NETWORK
TITLE = T-10.00 DOSE ON OFF
      O     "Blend to Preparation"."T-20".Raw_Material.Vinegar.DoseRun;
      O     "Blend to Preparation"."T-21".Raw_Material.Vinegar.DoseRun;
      O     "Blend to Preparation"."T-30".Raw_Material.Vinegar.DoseRun;
      O     "Blend to Preparation"."T-31".Raw_Material.Vinegar.DoseRun;
      O     "Blend to Preparation"."T-40".Raw_Material.Vinegar.DoseRun;
      O     "Blend to Preparation"."T-41".Raw_Material.Vinegar.DoseRun;
      O     "T-05_Tomato"."Vinegar Req";

      =     "T-10_Vinegar".IN_Dose_Run;

NETWORK
TITLE = T-10.00 DOSE PAUSE
      O     "Blend to Preparation"."T-20".Raw_Material.Vinegar.DoseHeld;
      O     "Blend to Preparation"."T-21".Raw_Material.Vinegar.DoseHeld;
      O     "Blend to Preparation"."T-30".Raw_Material.Vinegar.DoseHeld;
      O     "Blend to Preparation"."T-31".Raw_Material.Vinegar.DoseHeld;
      O     "Blend to Preparation"."T-40".Raw_Material.Vinegar.DoseHeld;
      O     "Blend to Preparation"."T-41".Raw_Material.Vinegar.DoseHeld;
      O     "T-05_Tomato".Dose_Vinegar.QHELD;

      =     "T-10_Vinegar".IN_Dose_Held;

NETWORK
TITLE = T-10.00 DOSE VALVE CMD
      O(;
      A     "Blend to Preparation"."T-20".Raw_Material.Vinegar.DoseRun;
      A     "Blend to Preparation"."T-20".Raw_Material.Vinegar.ValveCMD;
      );
      O(;
      A     "Blend to Preparation"."T-21".Raw_Material.Vinegar.DoseRun;
      A     "Blend to Preparation"."T-21".Raw_Material.Vinegar.ValveCMD;
      );
      O(;
      A     "Blend to Preparation"."T-30".Raw_Material.Vinegar.DoseRun;
      A     "Blend to Preparation"."T-30".Raw_Material.Vinegar.ValveCMD;
      );
      O(;
      A     "Blend to Preparation"."T-31".Raw_Material.Vinegar.DoseRun;
      A     "Blend to Preparation"."T-31".Raw_Material.Vinegar.ValveCMD;
      );
      O(;
      A     "Blend to Preparation"."T-40".Raw_Material.Vinegar.DoseRun;
      A     "Blend to Preparation"."T-40".Raw_Material.Vinegar.ValveCMD;
      );
      O(;
      A     "Blend to Preparation"."T-41".Raw_Material.Vinegar.DoseRun;
      A     "Blend to Preparation"."T-41".Raw_Material.Vinegar.ValveCMD;
      );
      O(;
      A     "T-05_Tomato"."Vinegar Req";
      A     "T-05_Tomato".Dose_Vinegar.V_CMD;
      );

      =     "T-10_Vinegar".IN_Dose_Valve_Cmd;



NETWORK
TITLE = T-10.00 DOSE Pump CMD
      O(;
      A     "Blend to Preparation"."T-20".Raw_Material.Vinegar.DoseRun;
      A     "Blend to Preparation"."T-20".Raw_Material.Vinegar.PumpCMD;
      );
      O(;
      A     "Blend to Preparation"."T-21".Raw_Material.Vinegar.DoseRun;
      A     "Blend to Preparation"."T-21".Raw_Material.Vinegar.PumpCMD;
      );
      O(;
      A     "Blend to Preparation"."T-30".Raw_Material.Vinegar.DoseRun;
      A     "Blend to Preparation"."T-30".Raw_Material.Vinegar.PumpCMD;
      );
      O(;
      A     "Blend to Preparation"."T-31".Raw_Material.Vinegar.DoseRun;
      A     "Blend to Preparation"."T-31".Raw_Material.Vinegar.PumpCMD;
      );
      O(;
      A     "Blend to Preparation"."T-40".Raw_Material.Vinegar.DoseRun;
      A     "Blend to Preparation"."T-40".Raw_Material.Vinegar.PumpCMD;
      );
      O(;
      A     "Blend to Preparation"."T-41".Raw_Material.Vinegar.DoseRun;
      A     "Blend to Preparation"."T-41".Raw_Material.Vinegar.PumpCMD;
      );
      O(;
      A     "T-05_Tomato"."Vinegar Req";
      A     "T-05_Tomato".Dose_Vinegar.P_CMD;
      );

      =     "T-10_Vinegar".IN_Dose_Pump_Cmd;



NETWORK
TITLE = T-10.00 DOSE PUMP SPEED
// Checking
      O     "Blend to Preparation"."T-20".Raw_Material.Vinegar.DoseRun;
      JC    SP_10_FROM_20;
      O     "Blend to Preparation"."T-21".Raw_Material.Vinegar.DoseRun;
      JC    SP_10_FROM_21;
      O     "Blend to Preparation"."T-30".Raw_Material.Vinegar.DoseRun;
      JC    SP_10_FROM_30;
      O     "Blend to Preparation"."T-31".Raw_Material.Vinegar.DoseRun;
      JC    SP_10_FROM_31;
      O     "Blend to Preparation"."T-40".Raw_Material.Vinegar.DoseRun;
      JC    SP_10_FROM_40;
      O     "Blend to Preparation"."T-41".Raw_Material.Vinegar.DoseRun;
      JC    SP_10_FROM_41;
      O     "T-05_Tomato"."Vinegar Req";
      JC    SP_10_FROM_Tomato;

//Jump to end if Blend not Dosing
      JC    SP_10_SELF;
//Load Set Point
SP_10_FROM_20:L     "Blend to Preparation".Recipe."T-20".Vinegar.SP_PumpSpeed;
      T     "T-10_Vinegar".IN_Dose_Pump_Sp;
      JC    SP_10_SELF;
SP_10_FROM_21:L     "Blend to Preparation".Recipe."T-21".Vinegar.SP_PumpSpeed;
      T     "T-10_Vinegar".IN_Dose_Pump_Sp;
      JC    SP_10_SELF;
SP_10_FROM_30:L     "Blend to Preparation".Recipe."T-30".Vinegar.SP_PumpSpeed;
      T     "T-10_Vinegar".IN_Dose_Pump_Sp;
      JC    SP_10_SELF;
SP_10_FROM_31:L     "Blend to Preparation".Recipe."T-31".Vinegar.SP_PumpSpeed;
      T     "T-10_Vinegar".IN_Dose_Pump_Sp;
      JC    SP_10_SELF;
SP_10_FROM_40:L     "Blend to Preparation".Recipe."T-40".Vinegar.SP_PumpSpeed;
      T     "T-10_Vinegar".IN_Dose_Pump_Sp;
      JC    SP_10_SELF;
SP_10_FROM_41:L     "Blend to Preparation".Recipe."T-41".Vinegar.SP_PumpSpeed;
      T     "T-10_Vinegar".IN_Dose_Pump_Sp;
      JC    SP_10_SELF;
SP_10_FROM_Tomato:L     "T-05_Tomato".Dose_Vinegar.P_SPEED;
      T     "T-10_Vinegar".IN_Dose_Pump_Sp;
      JC    SP_10_SELF;

// END
SP_10_SELF:L     "T-10_Vinegar".IN_Dose_Pump_Sp;
      T     "T-10_Vinegar".IN_Dose_Pump_Sp;


REGION Network 130: T-010.00 LineTransferOK
   RUNG wire#powerrail
      Contact( "AlwaysTRUE" )
      wire#w1
      Contact( "Blend to Preparation"."T-20".LineVinegar_OK )
      wire#w2
      Coil( "T-10_Vinegar".IN_Dose_LineOK )
   END_RUNG
   RUNG wire#w1
      Contact( "Blend to Preparation"."T-21".LineVinegar_OK )
   END_RUNG wire#w2
   RUNG wire#w1
      Contact( "Blend to Preparation"."T-30".LineVinegar_OK )
   END_RUNG wire#w2
   RUNG wire#w1
      Contact( "Blend to Preparation"."T-31".LineVinegar_OK )
   END_RUNG wire#w2
   RUNG wire#w1
      Contact( "Blend to Preparation"."T-40".LineVinegar_OK )
   END_RUNG wire#w2
   RUNG wire#w1
      Contact( "Blend to Preparation"."T-41".LineVinegar_OK )
   END_RUNG wire#w2
   RUNG wire#w1
      Contact( "T-05_Tomato".IN_FBAV_Vinegar )
   END_RUNG wire#w2
   // the same network as SCL:
   "T-10_Vinegar".IN_Dose_LineOK := "AlwaysTRUE" AND ("Blend to Preparation"."T-20".LineVinegar_OK OR "Blend to Preparation"."T-21".LineVinegar_OK OR "Blend to Preparation"."T-30".LineVinegar_OK OR "Blend to Preparation"."T-31".LineVinegar_OK OR "Blend to Preparation"."T-40".LineVinegar_OK OR "Blend to Preparation"."T-41".LineVinegar_OK OR "T-05_Tomato".IN_FBAV_Vinegar);
END_REGION

REGION Network 131: T-10.00____VINEGAR
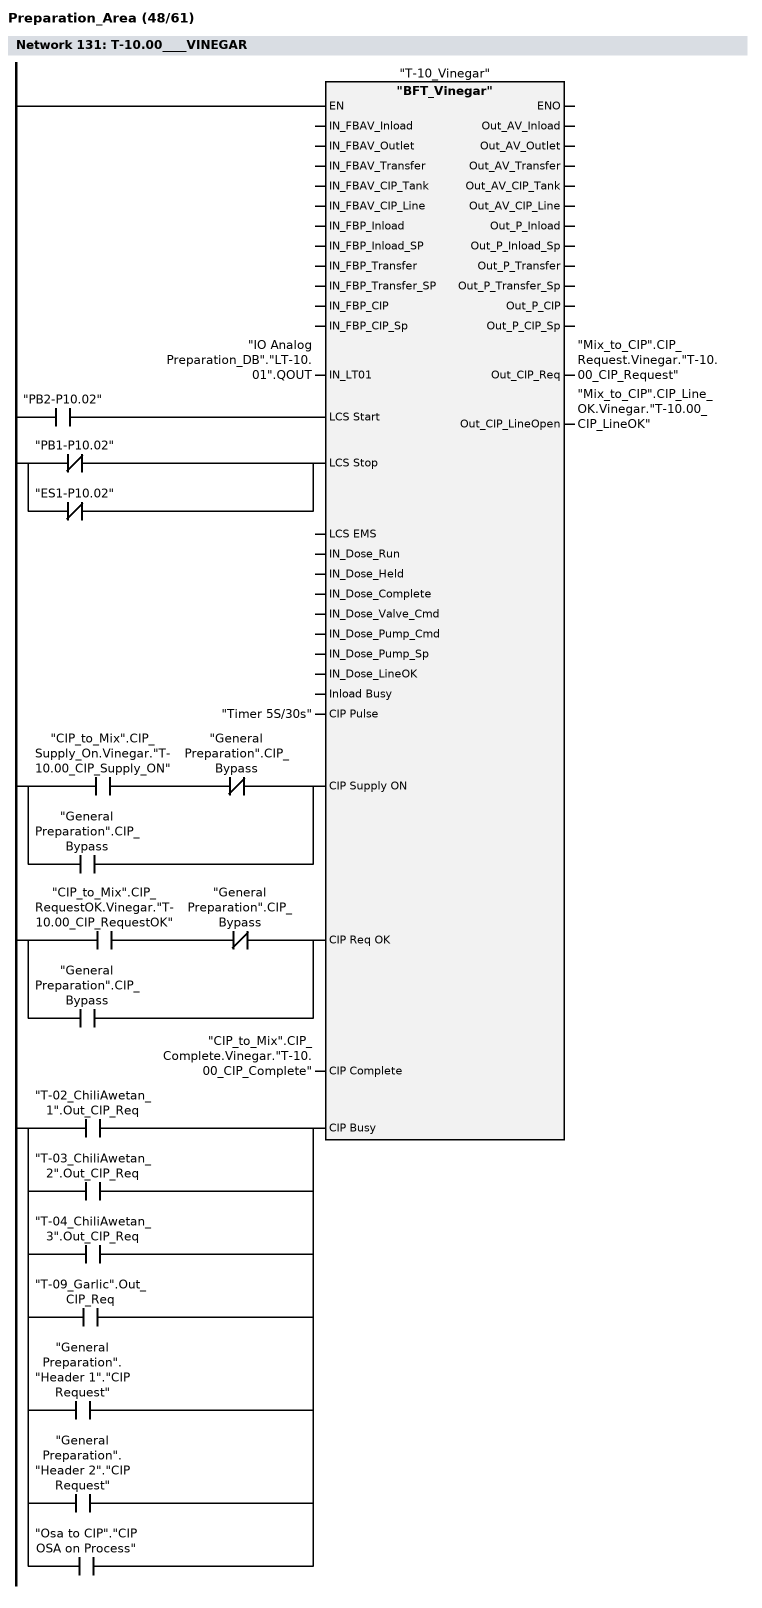
   RUNG wire#powerrail
      "T-10_Vinegar"("LCS Start" := wire#w1, "LCS Stop" := wire#w2, "CIP Supply ON" := wire#w3, "CIP Req OK" := wire#w4, "CIP Busy" := wire#w5, IN_FBAV_Inload :=, IN_FBAV_Outlet :=, IN_FBAV_Transfer :=, IN_FBAV_CIP_Tank :=, IN_FBAV_CIP_Line :=, IN_FBP_Inload :=, IN_FBP_Inload_SP :=, IN_FBP_Transfer :=, IN_FBP_Transfer_SP :=, IN_FBP_CIP :=, IN_FBP_CIP_Sp :=, IN_LT01 := "IO Analog Preparation_DB"."LT-10.01".QOUT, "LCS EMS" :=, IN_Dose_Run :=, IN_Dose_Held :=, IN_Dose_Complete :=, IN_Dose_Valve_Cmd :=, IN_Dose_Pump_Cmd :=, IN_Dose_Pump_Sp :=, IN_Dose_LineOK :=, "Inload Busy" :=, "CIP Pulse" := "Timer 5S/30s", "CIP Complete" := "CIP_to_Mix".CIP_Complete.Vinegar."T-10.00_CIP_Complete", Out_AV_Inload =>, Out_AV_Outlet =>, Out_AV_Transfer =>, Out_AV_CIP_Tank =>, Out_AV_CIP_Line =>, Out_P_Inload =>, Out_P_Inload_Sp =>, Out_P_Transfer =>, Out_P_Transfer_Sp =>, Out_P_CIP =>, Out_P_CIP_Sp =>, Out_CIP_Req => "Mix_to_CIP".CIP_Request.Vinegar."T-10.00_CIP_Request", Out_CIP_LineOpen => "Mix_to_CIP".CIP_Line_OK.Vinegar."T-10.00_CIP_LineOK")
   END_RUNG
   RUNG wire#powerrail
      Contact( "PB2-P10.02" )
   END_RUNG wire#w1
   RUNG wire#powerrail
      I_Contact( "PB1-P10.02" )
   END_RUNG wire#w2
   RUNG wire#powerrail
      I_Contact( "ES1-P10.02" )
   END_RUNG wire#w2
   RUNG wire#powerrail
      Contact( "CIP_to_Mix".CIP_Supply_On.Vinegar."T-10.00_CIP_Supply_ON" )
      I_Contact( "General Preparation".CIP_Bypass )
   END_RUNG wire#w3
   RUNG wire#powerrail
      Contact( "General Preparation".CIP_Bypass )
   END_RUNG wire#w3
   RUNG wire#powerrail
      Contact( "CIP_to_Mix".CIP_RequestOK.Vinegar."T-10.00_CIP_RequestOK" )
      I_Contact( "General Preparation".CIP_Bypass )
   END_RUNG wire#w4
   RUNG wire#powerrail
      Contact( "General Preparation".CIP_Bypass )
   END_RUNG wire#w4
   RUNG wire#powerrail
      Contact( "T-02_ChiliAwetan_1".Out_CIP_Req )
   END_RUNG wire#w5
   RUNG wire#powerrail
      Contact( "T-03_ChiliAwetan_2".Out_CIP_Req )
   END_RUNG wire#w5
   RUNG wire#powerrail
      Contact( "T-04_ChiliAwetan_3".Out_CIP_Req )
   END_RUNG wire#w5
   RUNG wire#powerrail
      Contact( "T-09_Garlic".Out_CIP_Req )
   END_RUNG wire#w5
   RUNG wire#powerrail
      Contact( "General Preparation"."Header 1"."CIP Request" )
   END_RUNG wire#w5
   RUNG wire#powerrail
      Contact( "General Preparation"."Header 2"."CIP Request" )
   END_RUNG wire#w5
   RUNG wire#powerrail
      Contact( "Osa to CIP"."CIP OSA on Process" )
   END_RUNG wire#w5
   // the same network as SCL:
   "T-10_Vinegar"(IN_LT01 := "IO Analog Preparation_DB"."LT-10.01".QOUT,   // "BFT_Vinegar"
                  "LCS Start" := "PB2-P10.02",
                  "LCS Stop" := NOT "PB1-P10.02" OR NOT "ES1-P10.02",
                  "CIP Pulse" := "Timer 5S/30s",
                  "CIP Supply ON" := ("CIP_to_Mix".CIP_Supply_On.Vinegar."T-10.00_CIP_Supply_ON" AND NOT "General Preparation".CIP_Bypass) OR "General Preparation".CIP_Bypass,
                  "CIP Req OK" := ("CIP_to_Mix".CIP_RequestOK.Vinegar."T-10.00_CIP_RequestOK" AND NOT "General Preparation".CIP_Bypass) OR "General Preparation".CIP_Bypass,
                  "CIP Complete" := "CIP_to_Mix".CIP_Complete.Vinegar."T-10.00_CIP_Complete",
                  "CIP Busy" := "T-02_ChiliAwetan_1".Out_CIP_Req OR "T-03_ChiliAwetan_2".Out_CIP_Req OR "T-04_ChiliAwetan_3".Out_CIP_Req OR "T-09_Garlic".Out_CIP_Req OR "General Preparation"."Header 1"."CIP Request" OR "General Preparation"."Header 2"."CIP Request" OR "Osa to CIP"."CIP OSA on Process",
                  Out_CIP_Req => "Mix_to_CIP".CIP_Request.Vinegar."T-10.00_CIP_Request",
                  Out_CIP_LineOpen => "Mix_to_CIP".CIP_Line_OK.Vinegar."T-10.00_CIP_LineOK");
END_REGION

REGION Network 132: T-10.00 Valve Cmd
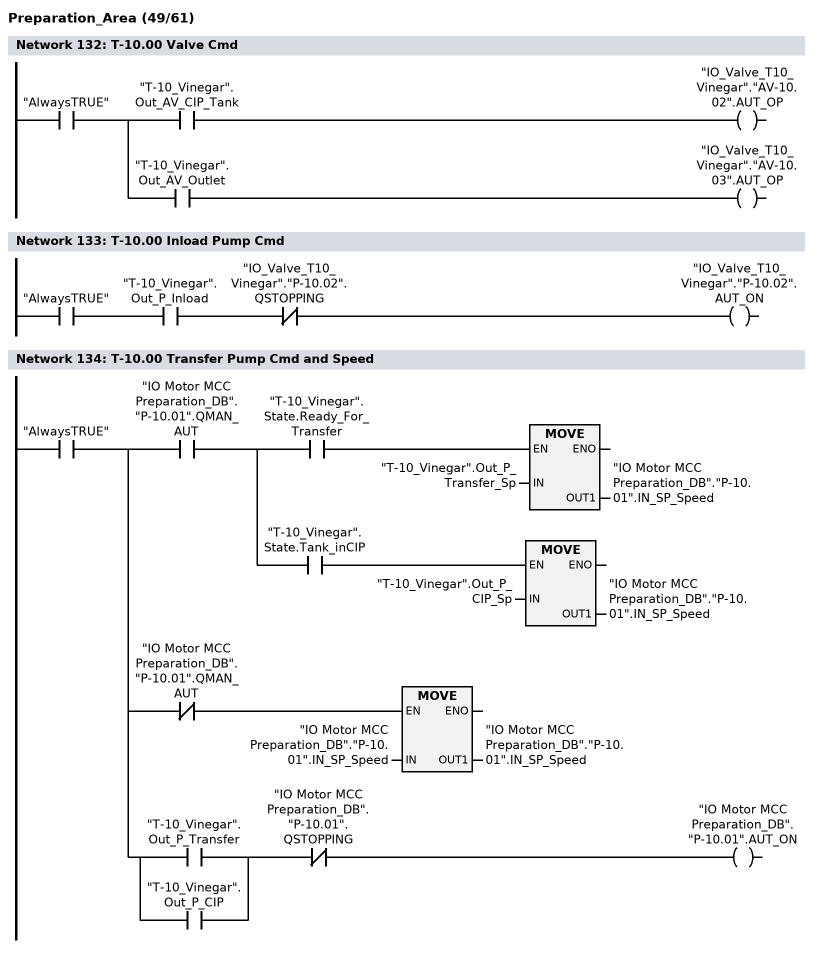
   RUNG wire#powerrail
      Contact( "AlwaysTRUE" )
      wire#w1
      Contact( "T-10_Vinegar".Out_AV_CIP_Tank )
      Coil( "IO_Valve_T10_Vinegar"."AV-10.02".AUT_OP )
   END_RUNG
   RUNG wire#w1
      Contact( "T-10_Vinegar".Out_AV_Outlet )
      Coil( "IO_Valve_T10_Vinegar"."AV-10.03".AUT_OP )
   END_RUNG
   // the same network as SCL:
   "IO_Valve_T10_Vinegar"."AV-10.02".AUT_OP := "AlwaysTRUE" AND "T-10_Vinegar".Out_AV_CIP_Tank;
   "IO_Valve_T10_Vinegar"."AV-10.03".AUT_OP := "AlwaysTRUE" AND "T-10_Vinegar".Out_AV_Outlet;
END_REGION

REGION Network 133: T-10.00 Inload Pump Cmd
   RUNG wire#powerrail
      Contact( "AlwaysTRUE" )
      Contact( "T-10_Vinegar".Out_P_Inload )
      I_Contact( "IO_Valve_T10_Vinegar"."P-10.02".QSTOPPING )
      Coil( "IO_Valve_T10_Vinegar"."P-10.02".AUT_ON )
   END_RUNG
   // the same network as SCL:
   "IO_Valve_T10_Vinegar"."P-10.02".AUT_ON := "AlwaysTRUE" AND "T-10_Vinegar".Out_P_Inload AND NOT "IO_Valve_T10_Vinegar"."P-10.02".QSTOPPING;
END_REGION

REGION Network 134: T-10.00 Transfer Pump Cmd and Speed
   RUNG wire#powerrail
      Contact( "AlwaysTRUE" )
      wire#w1
      Contact( "IO Motor MCC Preparation_DB"."P-10.01".QMAN_AUT )
      wire#w2
      Contact( "T-10_Vinegar".State.Ready_For_Transfer )
      Move(in := "T-10_Vinegar".Out_P_Transfer_Sp, out1 => "IO Motor MCC Preparation_DB"."P-10.01".IN_SP_Speed)
   END_RUNG
   RUNG wire#w2
      Contact( "T-10_Vinegar".State.Tank_inCIP )
      Move(in := "T-10_Vinegar".Out_P_CIP_Sp, out1 => "IO Motor MCC Preparation_DB"."P-10.01".IN_SP_Speed)
   END_RUNG
   RUNG wire#w1
      I_Contact( "IO Motor MCC Preparation_DB"."P-10.01".QMAN_AUT )
      Move(in := "IO Motor MCC Preparation_DB"."P-10.01".IN_SP_Speed, out1 => "IO Motor MCC Preparation_DB"."P-10.01".IN_SP_Speed)
   END_RUNG
   RUNG wire#w1
      Contact( "T-10_Vinegar".Out_P_Transfer )
      wire#w3
      I_Contact( "IO Motor MCC Preparation_DB"."P-10.01".QSTOPPING )
      Coil( "IO Motor MCC Preparation_DB"."P-10.01".AUT_ON )
   END_RUNG
   RUNG wire#w1
      Contact( "T-10_Vinegar".Out_P_CIP )
   END_RUNG wire#w3
   // the same network as SCL:
   #_w1 := "AlwaysTRUE" AND "IO Motor MCC Preparation_DB"."P-10.01".QMAN_AUT;
   IF #_w1 AND "T-10_Vinegar".State.Ready_For_Transfer THEN
       "IO Motor MCC Preparation_DB"."P-10.01".IN_SP_Speed := "T-10_Vinegar".Out_P_Transfer_Sp;
   END_IF;
   IF #_w1 AND "T-10_Vinegar".State.Tank_inCIP THEN
       "IO Motor MCC Preparation_DB"."P-10.01".IN_SP_Speed := "T-10_Vinegar".Out_P_CIP_Sp;
   END_IF;
   IF "AlwaysTRUE" AND NOT "IO Motor MCC Preparation_DB"."P-10.01".QMAN_AUT THEN
       "IO Motor MCC Preparation_DB"."P-10.01".IN_SP_Speed := "IO Motor MCC Preparation_DB"."P-10.01".IN_SP_Speed;
   END_IF;
   "IO Motor MCC Preparation_DB"."P-10.01".AUT_ON := "AlwaysTRUE" AND ("T-10_Vinegar".Out_P_Transfer OR "T-10_Vinegar".Out_P_CIP) AND NOT "IO Motor MCC Preparation_DB"."P-10.01".QSTOPPING;
END_REGION

REGION Network 135: T-10.00 Feedback Instrument
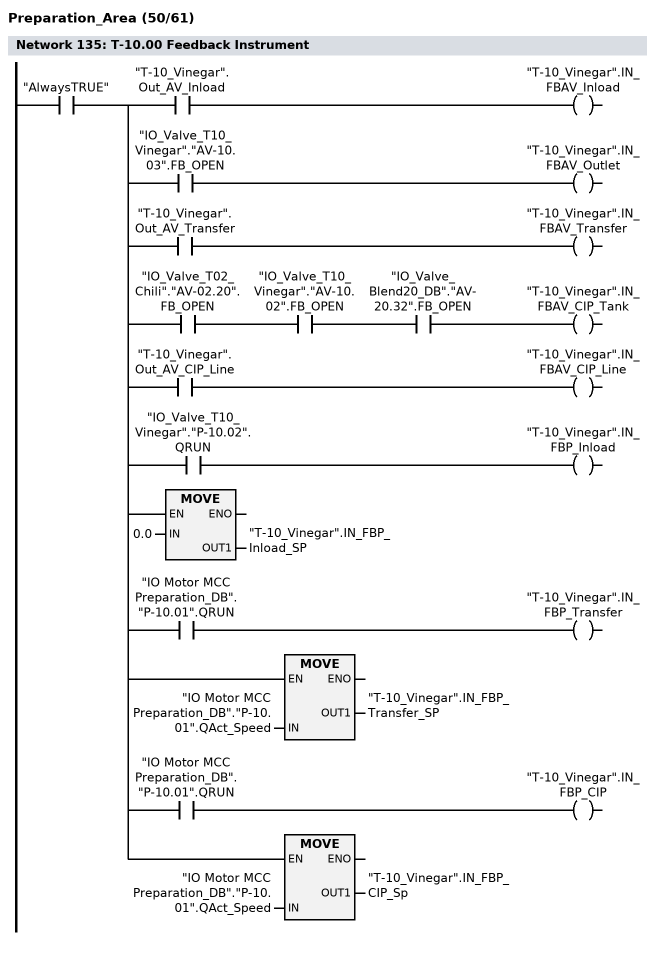
   RUNG wire#powerrail
      Contact( "AlwaysTRUE" )
      wire#w1
      Contact( "T-10_Vinegar".Out_AV_Inload )
      Coil( "T-10_Vinegar".IN_FBAV_Inload )
   END_RUNG
   RUNG wire#w1
      Contact( "IO_Valve_T10_Vinegar"."AV-10.03".FB_OPEN )
      Coil( "T-10_Vinegar".IN_FBAV_Outlet )
   END_RUNG
   RUNG wire#w1
      Contact( "T-10_Vinegar".Out_AV_Transfer )
      Coil( "T-10_Vinegar".IN_FBAV_Transfer )
   END_RUNG
   RUNG wire#w1
      Contact( "IO_Valve_T02_Chili"."AV-02.20".FB_OPEN )
      Contact( "IO_Valve_T10_Vinegar"."AV-10.02".FB_OPEN )
      Contact( "IO_Valve_Blend20_DB"."AV-20.32".FB_OPEN )
      Coil( "T-10_Vinegar".IN_FBAV_CIP_Tank )
   END_RUNG
   RUNG wire#w1
      Contact( "T-10_Vinegar".Out_AV_CIP_Line )
      Coil( "T-10_Vinegar".IN_FBAV_CIP_Line )
   END_RUNG
   RUNG wire#w1
      Contact( "IO_Valve_T10_Vinegar"."P-10.02".QRUN )
      Coil( "T-10_Vinegar".IN_FBP_Inload )
   END_RUNG
   RUNG wire#w1
      Move(in := 0.0, out1 => "T-10_Vinegar".IN_FBP_Inload_SP)
   END_RUNG
   RUNG wire#w1
      Contact( "IO Motor MCC Preparation_DB"."P-10.01".QRUN )
      Coil( "T-10_Vinegar".IN_FBP_Transfer )
   END_RUNG
   RUNG wire#w1
      Move(in := "IO Motor MCC Preparation_DB"."P-10.01".QAct_Speed, out1 => "T-10_Vinegar".IN_FBP_Transfer_SP)
   END_RUNG
   RUNG wire#w1
      Contact( "IO Motor MCC Preparation_DB"."P-10.01".QRUN )
      Coil( "T-10_Vinegar".IN_FBP_CIP )
   END_RUNG
   RUNG wire#w1
      Move(in := "IO Motor MCC Preparation_DB"."P-10.01".QAct_Speed, out1 => "T-10_Vinegar".IN_FBP_CIP_Sp)
   END_RUNG
   // the same network as SCL:
   "T-10_Vinegar".IN_FBAV_Inload := "AlwaysTRUE" AND "T-10_Vinegar".Out_AV_Inload;
   "T-10_Vinegar".IN_FBAV_Outlet := "AlwaysTRUE" AND "IO_Valve_T10_Vinegar"."AV-10.03".FB_OPEN;
   "T-10_Vinegar".IN_FBAV_Transfer := "AlwaysTRUE" AND "T-10_Vinegar".Out_AV_Transfer;
   "T-10_Vinegar".IN_FBAV_CIP_Tank := "AlwaysTRUE" AND "IO_Valve_T02_Chili"."AV-02.20".FB_OPEN AND "IO_Valve_T10_Vinegar"."AV-10.02".FB_OPEN AND "IO_Valve_Blend20_DB"."AV-20.32".FB_OPEN;
   "T-10_Vinegar".IN_FBAV_CIP_Line := "AlwaysTRUE" AND "T-10_Vinegar".Out_AV_CIP_Line;
   "T-10_Vinegar".IN_FBP_Inload := "AlwaysTRUE" AND "IO_Valve_T10_Vinegar"."P-10.02".QRUN;
   IF "AlwaysTRUE" THEN "T-10_Vinegar".IN_FBP_Inload_SP := 0.0; END_IF;
   "T-10_Vinegar".IN_FBP_Transfer := "AlwaysTRUE" AND "IO Motor MCC Preparation_DB"."P-10.01".QRUN;
   IF "AlwaysTRUE" THEN
       "T-10_Vinegar".IN_FBP_Transfer_SP := "IO Motor MCC Preparation_DB"."P-10.01".QAct_Speed;
   END_IF;
   "T-10_Vinegar".IN_FBP_CIP := "AlwaysTRUE" AND "IO Motor MCC Preparation_DB"."P-10.01".QRUN;
   IF "AlwaysTRUE" THEN
       "T-10_Vinegar".IN_FBP_CIP_Sp := "IO Motor MCC Preparation_DB"."P-10.01".QAct_Speed;
   END_IF;
END_REGION

REGION Network 136: T-10.00 Comm to Blend
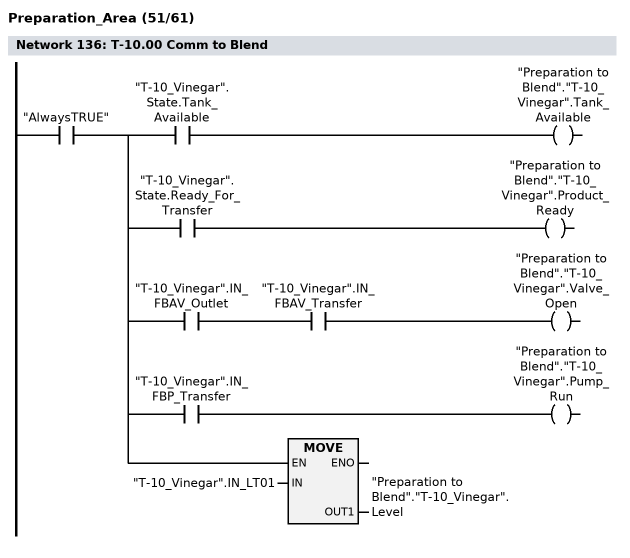
   RUNG wire#powerrail
      Contact( "AlwaysTRUE" )
      wire#w1
      Contact( "T-10_Vinegar".State.Tank_Available )
      Coil( "Preparation to Blend"."T-10_Vinegar".Tank_Available )
   END_RUNG
   RUNG wire#w1
      Contact( "T-10_Vinegar".State.Ready_For_Transfer )
      Coil( "Preparation to Blend"."T-10_Vinegar".Product_Ready )
   END_RUNG
   RUNG wire#w1
      Contact( "T-10_Vinegar".IN_FBAV_Outlet )
      Contact( "T-10_Vinegar".IN_FBAV_Transfer )
      Coil( "Preparation to Blend"."T-10_Vinegar".Valve_Open )
   END_RUNG
   RUNG wire#w1
      Contact( "T-10_Vinegar".IN_FBP_Transfer )
      Coil( "Preparation to Blend"."T-10_Vinegar".Pump_Run )
   END_RUNG
   RUNG wire#w1
      Move(in := "T-10_Vinegar".IN_LT01, out1 => "Preparation to Blend"."T-10_Vinegar".Level)
   END_RUNG
   // the same network as SCL:
   "Preparation to Blend"."T-10_Vinegar".Tank_Available := "AlwaysTRUE" AND "T-10_Vinegar".State.Tank_Available;
   "Preparation to Blend"."T-10_Vinegar".Product_Ready := "AlwaysTRUE" AND "T-10_Vinegar".State.Ready_For_Transfer;
   "Preparation to Blend"."T-10_Vinegar".Valve_Open := "AlwaysTRUE" AND "T-10_Vinegar".IN_FBAV_Outlet AND "T-10_Vinegar".IN_FBAV_Transfer;
   "Preparation to Blend"."T-10_Vinegar".Pump_Run := "AlwaysTRUE" AND "T-10_Vinegar".IN_FBP_Transfer;
   IF "AlwaysTRUE" THEN "Preparation to Blend"."T-10_Vinegar".Level := "T-10_Vinegar".IN_LT01; END_IF;
END_REGION

NETWORK
TITLE = T-51.00 DOSE ON OFF
      O     "Blend to Preparation"."T-20".Raw_Material.HW.DoseRun;
      O     "Blend to Preparation"."T-21".Raw_Material.HW.DoseRun;
      O     "Blend to Preparation"."T-30".Raw_Material.HW.DoseRun;
      O     "Blend to Preparation"."T-31".Raw_Material.HW.DoseRun;
      O     "Blend to Preparation"."T-40".Raw_Material.HW.DoseRun;
      O     "Blend to Preparation"."T-41".Raw_Material.HW.DoseRun;
      =     "T-51_HW".IN_Dose_Run;

NETWORK
TITLE = T-51.00 DOSE PAUSE
      O     "Blend to Preparation"."T-20".Raw_Material.HW.DoseHeld;
      O     "Blend to Preparation"."T-21".Raw_Material.HW.DoseHeld;
      O     "Blend to Preparation"."T-30".Raw_Material.HW.DoseHeld;
      O     "Blend to Preparation"."T-31".Raw_Material.HW.DoseHeld;
      O     "Blend to Preparation"."T-40".Raw_Material.HW.DoseHeld;
      O     "Blend to Preparation"."T-41".Raw_Material.HW.DoseHeld;
      =     "T-51_HW".IN_Dose_Held;

NETWORK
TITLE = T-51.00 DOSE VALVE CMD
      O(;
      A     "Blend to Preparation"."T-20".Raw_Material.HW.DoseRun;
      A     "Blend to Preparation"."T-20".Raw_Material.HW.ValveCMD;
      );
      O(;
      A     "Blend to Preparation"."T-21".Raw_Material.HW.DoseRun;
      A     "Blend to Preparation"."T-21".Raw_Material.HW.ValveCMD;
      );
      O(;
      A     "Blend to Preparation"."T-30".Raw_Material.HW.DoseRun;
      A     "Blend to Preparation"."T-30".Raw_Material.HW.ValveCMD;
      );
      O(;
      A     "Blend to Preparation"."T-31".Raw_Material.HW.DoseRun;
      A     "Blend to Preparation"."T-31".Raw_Material.HW.ValveCMD;
      );
      O(;
      A     "Blend to Preparation"."T-40".Raw_Material.HW.DoseRun;
      A     "Blend to Preparation"."T-40".Raw_Material.HW.ValveCMD;
      );
      O(;
      A     "Blend to Preparation"."T-41".Raw_Material.HW.DoseRun;
      A     "Blend to Preparation"."T-41".Raw_Material.HW.ValveCMD;
      );
      =     "T-51_HW".IN_Dose_Valve_Cmd;

NETWORK
TITLE = T-51.00 DOSE Pump CMD
      O(;
      A     "Blend to Preparation"."T-20".Raw_Material.HW.DoseRun;
      A     "Blend to Preparation"."T-20".Raw_Material.HW.PumpCMD;
      );
      O(;
      A     "Blend to Preparation"."T-21".Raw_Material.HW.DoseRun;
      A     "Blend to Preparation"."T-21".Raw_Material.HW.PumpCMD;
      );
      O(;
      A     "Blend to Preparation"."T-30".Raw_Material.HW.DoseRun;
      A     "Blend to Preparation"."T-30".Raw_Material.HW.PumpCMD;
      );
      O(;
      A     "Blend to Preparation"."T-31".Raw_Material.HW.DoseRun;
      A     "Blend to Preparation"."T-31".Raw_Material.HW.PumpCMD;
      );
      O(;
      A     "Blend to Preparation"."T-40".Raw_Material.HW.DoseRun;
      A     "Blend to Preparation"."T-40".Raw_Material.HW.PumpCMD;
      );
      O(;
      A     "Blend to Preparation"."T-41".Raw_Material.HW.DoseRun;
      A     "Blend to Preparation"."T-41".Raw_Material.HW.PumpCMD;
      );
      =     "T-51_HW".IN_Dose_Pump_Cmd;

NETWORK
TITLE = T-51.00 DOSE PUMP SPEED
// Checking
      O     "Blend to Preparation"."T-20".Raw_Material.HW.DoseRun;
      JC    SP_51_FROM_20;
      O     "Blend to Preparation"."T-21".Raw_Material.HW.DoseRun;
      JC    SP_51_FROM_21;
      O     "Blend to Preparation"."T-30".Raw_Material.HW.DoseRun;
      JC    SP_51_FROM_30;
      O     "Blend to Preparation"."T-31".Raw_Material.HW.DoseRun;
      JC    SP_51_FROM_31;
      O     "Blend to Preparation"."T-40".Raw_Material.HW.DoseRun;
      JC    SP_51_FROM_40;
      O     "Blend to Preparation"."T-41".Raw_Material.HW.DoseRun;
      JC    SP_51_FROM_41;
//Jump to end if Blend not Dosing
      JC    SP_51_SELF;
//Load Set Point
SP_51_FROM_20:L     "Blend to Preparation".Recipe."T-20".HW.SP_PumpSpeed;
      T     "T-51_HW".IN_Dose_Pump_Sp;
      JC    SP_51_SELF;
SP_51_FROM_21:L     "Blend to Preparation".Recipe."T-21".HW.SP_PumpSpeed;
      T     "T-51_HW".IN_Dose_Pump_Sp;
      JC    SP_51_SELF;
SP_51_FROM_30:L     "Blend to Preparation".Recipe."T-30".HW.SP_PumpSpeed;
      T     "T-51_HW".IN_Dose_Pump_Sp;
      JC    SP_51_SELF;
SP_51_FROM_31:L     "Blend to Preparation".Recipe."T-31".HW.SP_PumpSpeed;
      T     "T-51_HW".IN_Dose_Pump_Sp;
      JC    SP_51_SELF;
SP_51_FROM_40:L     "Blend to Preparation".Recipe."T-40".HW.SP_PumpSpeed;
      T     "T-51_HW".IN_Dose_Pump_Sp;
      JC    SP_51_SELF;
SP_51_FROM_41:L     "Blend to Preparation".Recipe."T-41".HW.SP_PumpSpeed;
      T     "T-51_HW".IN_Dose_Pump_Sp;
      JC    SP_51_SELF;
// END
SP_51_SELF:L     "T-51_HW".IN_Dose_Pump_Sp;
      T     "T-51_HW".IN_Dose_Pump_Sp;

NETWORK
TITLE = T-51.00 Header Req
// HEADER 1 Req
      O     "Blend to Preparation"."T-20".Raw_Material.HW.Header1_Req;
      O     "Blend to Preparation"."T-21".Raw_Material.HW.Header1_Req;
      O     "Blend to Preparation"."T-30".Raw_Material.HW.Header1_Req;
      O     "Blend to Preparation"."T-31".Raw_Material.HW.Header1_Req;
      O     "Blend to Preparation"."T-40".Raw_Material.HW.Header1_Req;
      O     "Blend to Preparation"."T-41".Raw_Material.HW.Header1_Req;
      =     "T-51_HW".IN_Dose_Header_1;

// HEADER 2 Req
      O     "Blend to Preparation"."T-20".Raw_Material.HW.Header2_Req;
      O     "Blend to Preparation"."T-21".Raw_Material.HW.Header2_Req;
      O     "Blend to Preparation"."T-30".Raw_Material.HW.Header2_Req;
      O     "Blend to Preparation"."T-31".Raw_Material.HW.Header2_Req;
      O     "Blend to Preparation"."T-40".Raw_Material.HW.Header2_Req;
      O     "Blend to Preparation"."T-41".Raw_Material.HW.Header2_Req;
      =     "T-51_HW".IN_Dose_Header_2;

REGION Network 145: T-51.00 LineTransferOK
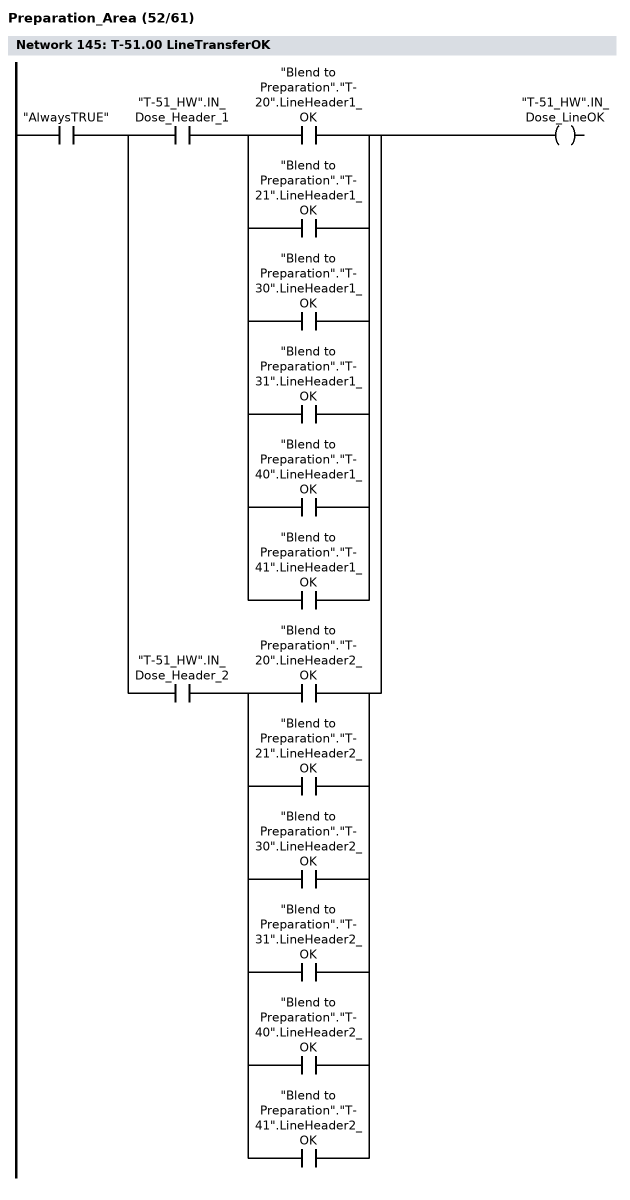
   RUNG wire#powerrail
      Contact( "AlwaysTRUE" )
      wire#w1
      Contact( "T-51_HW".IN_Dose_Header_1 )
      wire#w2
      Contact( "Blend to Preparation"."T-20".LineHeader1_OK )
      wire#w3
      Coil( "T-51_HW".IN_Dose_LineOK )
   END_RUNG
   RUNG wire#w2
      Contact( "Blend to Preparation"."T-21".LineHeader1_OK )
   END_RUNG wire#w3
   RUNG wire#w2
      Contact( "Blend to Preparation"."T-30".LineHeader1_OK )
   END_RUNG wire#w3
   RUNG wire#w2
      Contact( "Blend to Preparation"."T-31".LineHeader1_OK )
   END_RUNG wire#w3
   RUNG wire#w2
      Contact( "Blend to Preparation"."T-40".LineHeader1_OK )
   END_RUNG wire#w3
   RUNG wire#w2
      Contact( "Blend to Preparation"."T-41".LineHeader1_OK )
   END_RUNG wire#w3
   RUNG wire#w1
      Contact( "T-51_HW".IN_Dose_Header_2 )
      wire#w4
      Contact( "Blend to Preparation"."T-20".LineHeader2_OK )
   END_RUNG wire#w3
   RUNG wire#w4
      Contact( "Blend to Preparation"."T-21".LineHeader2_OK )
   END_RUNG wire#w3
   RUNG wire#w4
      Contact( "Blend to Preparation"."T-30".LineHeader2_OK )
   END_RUNG wire#w3
   RUNG wire#w4
      Contact( "Blend to Preparation"."T-31".LineHeader2_OK )
   END_RUNG wire#w3
   RUNG wire#w4
      Contact( "Blend to Preparation"."T-40".LineHeader2_OK )
   END_RUNG wire#w3
   RUNG wire#w4
      Contact( "Blend to Preparation"."T-41".LineHeader2_OK )
   END_RUNG wire#w3
   // the same network as SCL:
   "T-51_HW".IN_Dose_LineOK := "AlwaysTRUE" AND (("T-51_HW".IN_Dose_Header_1 AND ("Blend to Preparation"."T-20".LineHeader1_OK OR "Blend to Preparation"."T-21".LineHeader1_OK OR "Blend to Preparation"."T-30".LineHeader1_OK OR "Blend to Preparation"."T-31".LineHeader1_OK OR "Blend to Preparation"."T-40".LineHeader1_OK OR "Blend to Preparation"."T-41".LineHeader1_OK)) OR ("T-51_HW".IN_Dose_Header_2 AND ("Blend to Preparation"."T-20".LineHeader2_OK OR "Blend to Preparation"."T-21".LineHeader2_OK OR "Blend to Preparation"."T-30".LineHeader2_OK OR "Blend to Preparation"."T-31".LineHeader2_OK OR "Blend to Preparation"."T-40".LineHeader2_OK OR "Blend to Preparation"."T-41".LineHeader2_OK)));
END_REGION

REGION Network 146: T-51.01 Hot Water
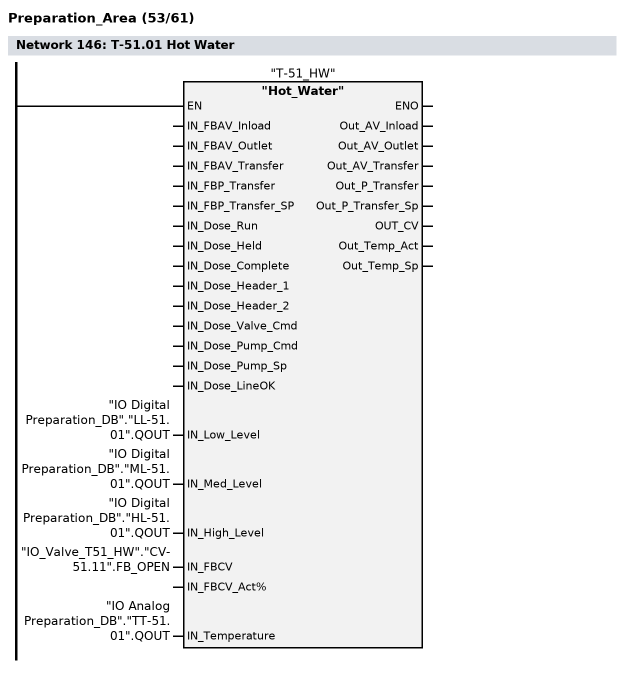
   RUNG wire#powerrail
      "T-51_HW"(IN_FBAV_Inload :=, IN_FBAV_Outlet :=, IN_FBAV_Transfer :=, IN_FBP_Transfer :=, IN_FBP_Transfer_SP :=, IN_Dose_Run :=, IN_Dose_Held :=, IN_Dose_Complete :=, IN_Dose_Header_1 :=, IN_Dose_Header_2 :=, IN_Dose_Valve_Cmd :=, IN_Dose_Pump_Cmd :=, IN_Dose_Pump_Sp :=, IN_Dose_LineOK :=, IN_Low_Level := "IO Digital Preparation_DB"."LL-51.01".QOUT, IN_Med_Level := "IO Digital Preparation_DB"."ML-51.01".QOUT, IN_High_Level := "IO Digital Preparation_DB"."HL-51.01".QOUT, IN_FBCV := "IO_Valve_T51_HW"."CV-51.11".FB_OPEN, "IN_FBCV_Act%" :=, IN_Temperature := "IO Analog Preparation_DB"."TT-51.01".QOUT, Out_AV_Inload =>, Out_AV_Outlet =>, Out_AV_Transfer =>, Out_P_Transfer =>, Out_P_Transfer_Sp =>, OUT_CV =>, Out_Temp_Act =>, Out_Temp_Sp =>)
   END_RUNG
   // the same network as SCL:
   "T-51_HW"(IN_Low_Level := "IO Digital Preparation_DB"."LL-51.01".QOUT,   // "Hot_Water"
             IN_Med_Level := "IO Digital Preparation_DB"."ML-51.01".QOUT,
             IN_High_Level := "IO Digital Preparation_DB"."HL-51.01".QOUT,
             IN_FBCV := "IO_Valve_T51_HW"."CV-51.11".FB_OPEN,
             IN_Temperature := "IO Analog Preparation_DB"."TT-51.01".QOUT);
END_REGION

REGION Network 147: T-51.00 Valve Cmd
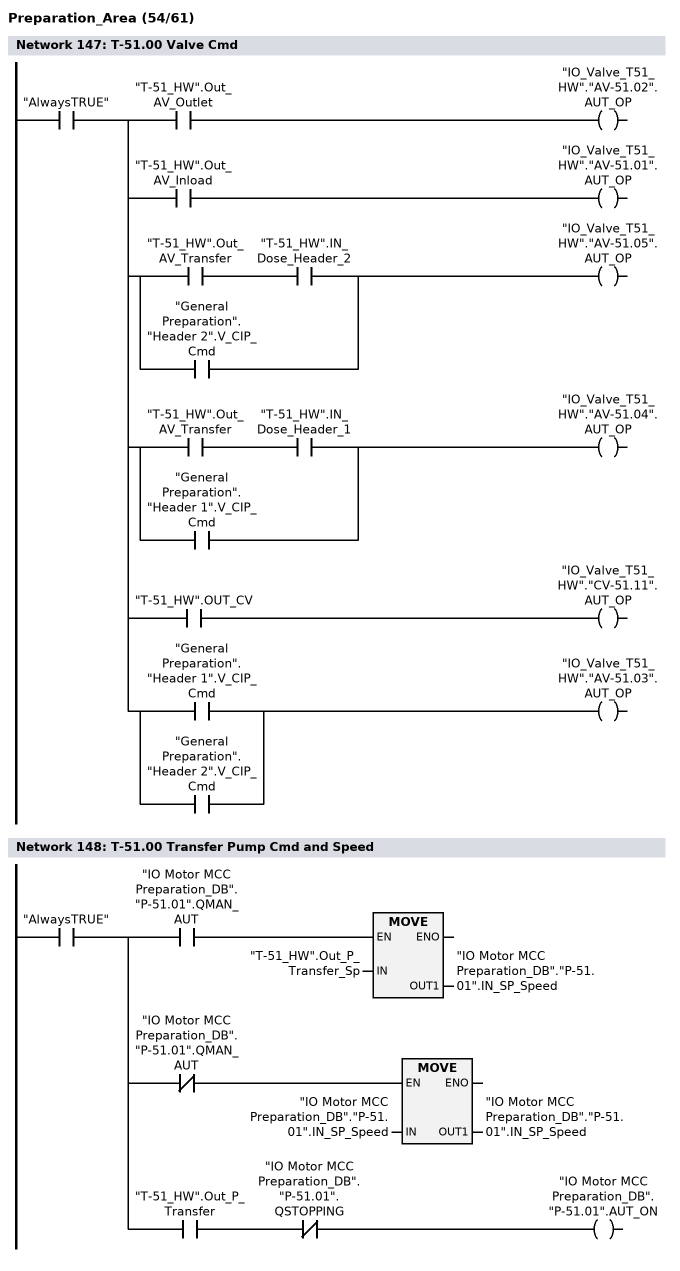
   RUNG wire#powerrail
      Contact( "AlwaysTRUE" )
      wire#w1
      Contact( "T-51_HW".Out_AV_Outlet )
      Coil( "IO_Valve_T51_HW"."AV-51.02".AUT_OP )
   END_RUNG
   RUNG wire#w1
      Contact( "T-51_HW".Out_AV_Inload )
      Coil( "IO_Valve_T51_HW"."AV-51.01".AUT_OP )
   END_RUNG
   RUNG wire#w1
      Contact( "T-51_HW".Out_AV_Transfer )
      Contact( "T-51_HW".IN_Dose_Header_2 )
      wire#w2
      Coil( "IO_Valve_T51_HW"."AV-51.05".AUT_OP )
   END_RUNG
   RUNG wire#w1
      Contact( "General Preparation"."Header 2".V_CIP_Cmd )
   END_RUNG wire#w2
   RUNG wire#w1
      Contact( "T-51_HW".Out_AV_Transfer )
      Contact( "T-51_HW".IN_Dose_Header_1 )
      wire#w3
      Coil( "IO_Valve_T51_HW"."AV-51.04".AUT_OP )
   END_RUNG
   RUNG wire#w1
      Contact( "General Preparation"."Header 1".V_CIP_Cmd )
   END_RUNG wire#w3
   RUNG wire#w1
      Contact( "T-51_HW".OUT_CV )
      Coil( "IO_Valve_T51_HW"."CV-51.11".AUT_OP )
   END_RUNG
   RUNG wire#w1
      Contact( "General Preparation"."Header 1".V_CIP_Cmd )
      wire#w4
      Coil( "IO_Valve_T51_HW"."AV-51.03".AUT_OP )
   END_RUNG
   RUNG wire#w1
      Contact( "General Preparation"."Header 2".V_CIP_Cmd )
   END_RUNG wire#w4
   // the same network as SCL:
   "IO_Valve_T51_HW"."AV-51.02".AUT_OP := "AlwaysTRUE" AND "T-51_HW".Out_AV_Outlet;
   "IO_Valve_T51_HW"."AV-51.01".AUT_OP := "AlwaysTRUE" AND "T-51_HW".Out_AV_Inload;
   "IO_Valve_T51_HW"."AV-51.05".AUT_OP := "AlwaysTRUE" AND (("T-51_HW".Out_AV_Transfer AND "T-51_HW".IN_Dose_Header_2) OR "General Preparation"."Header 2".V_CIP_Cmd);
   "IO_Valve_T51_HW"."AV-51.04".AUT_OP := "AlwaysTRUE" AND (("T-51_HW".Out_AV_Transfer AND "T-51_HW".IN_Dose_Header_1) OR "General Preparation"."Header 1".V_CIP_Cmd);
   "IO_Valve_T51_HW"."CV-51.11".AUT_OP := "AlwaysTRUE" AND "T-51_HW".OUT_CV;
   "IO_Valve_T51_HW"."AV-51.03".AUT_OP := "AlwaysTRUE" AND ("General Preparation"."Header 1".V_CIP_Cmd OR "General Preparation"."Header 2".V_CIP_Cmd);
END_REGION

REGION Network 148: T-51.00 Transfer Pump Cmd and Speed
   RUNG wire#powerrail
      Contact( "AlwaysTRUE" )
      wire#w1
      Contact( "IO Motor MCC Preparation_DB"."P-51.01".QMAN_AUT )
      Move(in := "T-51_HW".Out_P_Transfer_Sp, out1 => "IO Motor MCC Preparation_DB"."P-51.01".IN_SP_Speed)
   END_RUNG
   RUNG wire#w1
      I_Contact( "IO Motor MCC Preparation_DB"."P-51.01".QMAN_AUT )
      Move(in := "IO Motor MCC Preparation_DB"."P-51.01".IN_SP_Speed, out1 => "IO Motor MCC Preparation_DB"."P-51.01".IN_SP_Speed)
   END_RUNG
   RUNG wire#w1
      Contact( "T-51_HW".Out_P_Transfer )
      I_Contact( "IO Motor MCC Preparation_DB"."P-51.01".QSTOPPING )
      Coil( "IO Motor MCC Preparation_DB"."P-51.01".AUT_ON )
   END_RUNG
   // the same network as SCL:
   IF "AlwaysTRUE" AND "IO Motor MCC Preparation_DB"."P-51.01".QMAN_AUT THEN
       "IO Motor MCC Preparation_DB"."P-51.01".IN_SP_Speed := "T-51_HW".Out_P_Transfer_Sp;
   END_IF;
   IF "AlwaysTRUE" AND NOT "IO Motor MCC Preparation_DB"."P-51.01".QMAN_AUT THEN
       "IO Motor MCC Preparation_DB"."P-51.01".IN_SP_Speed := "IO Motor MCC Preparation_DB"."P-51.01".IN_SP_Speed;
   END_IF;
   "IO Motor MCC Preparation_DB"."P-51.01".AUT_ON := "AlwaysTRUE" AND "T-51_HW".Out_P_Transfer AND NOT "IO Motor MCC Preparation_DB"."P-51.01".QSTOPPING;
END_REGION

REGION Network 149: T-51.00 Feedback Instrument
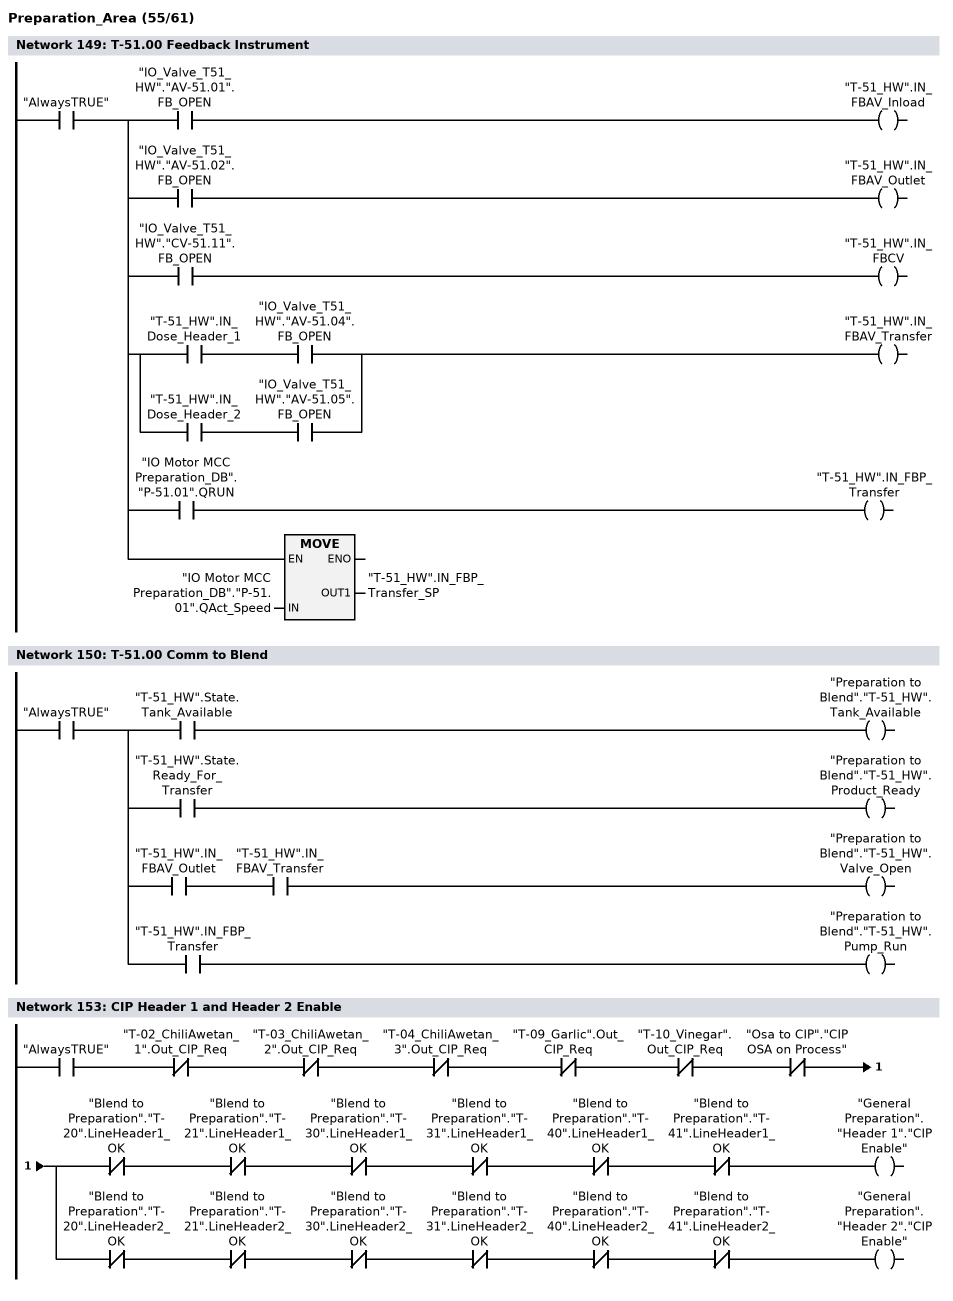
   RUNG wire#powerrail
      Contact( "AlwaysTRUE" )
      wire#w1
      Contact( "IO_Valve_T51_HW"."AV-51.01".FB_OPEN )
      Coil( "T-51_HW".IN_FBAV_Inload )
   END_RUNG
   RUNG wire#w1
      Contact( "IO_Valve_T51_HW"."AV-51.02".FB_OPEN )
      Coil( "T-51_HW".IN_FBAV_Outlet )
   END_RUNG
   RUNG wire#w1
      Contact( "IO_Valve_T51_HW"."CV-51.11".FB_OPEN )
      Coil( "T-51_HW".IN_FBCV )
   END_RUNG
   RUNG wire#w1
      Contact( "T-51_HW".IN_Dose_Header_1 )
      Contact( "IO_Valve_T51_HW"."AV-51.04".FB_OPEN )
      wire#w2
      Coil( "T-51_HW".IN_FBAV_Transfer )
   END_RUNG
   RUNG wire#w1
      Contact( "T-51_HW".IN_Dose_Header_2 )
      Contact( "IO_Valve_T51_HW"."AV-51.05".FB_OPEN )
   END_RUNG wire#w2
   RUNG wire#w1
      Contact( "IO Motor MCC Preparation_DB"."P-51.01".QRUN )
      Coil( "T-51_HW".IN_FBP_Transfer )
   END_RUNG
   RUNG wire#w1
      Move(in := "IO Motor MCC Preparation_DB"."P-51.01".QAct_Speed, out1 => "T-51_HW".IN_FBP_Transfer_SP)
   END_RUNG
   // the same network as SCL:
   "T-51_HW".IN_FBAV_Inload := "AlwaysTRUE" AND "IO_Valve_T51_HW"."AV-51.01".FB_OPEN;
   "T-51_HW".IN_FBAV_Outlet := "AlwaysTRUE" AND "IO_Valve_T51_HW"."AV-51.02".FB_OPEN;
   "T-51_HW".IN_FBCV := "AlwaysTRUE" AND "IO_Valve_T51_HW"."CV-51.11".FB_OPEN;
   "T-51_HW".IN_FBAV_Transfer := "AlwaysTRUE" AND (("T-51_HW".IN_Dose_Header_1 AND "IO_Valve_T51_HW"."AV-51.04".FB_OPEN) OR ("T-51_HW".IN_Dose_Header_2 AND "IO_Valve_T51_HW"."AV-51.05".FB_OPEN));
   "T-51_HW".IN_FBP_Transfer := "AlwaysTRUE" AND "IO Motor MCC Preparation_DB"."P-51.01".QRUN;
   IF "AlwaysTRUE" THEN
       "T-51_HW".IN_FBP_Transfer_SP := "IO Motor MCC Preparation_DB"."P-51.01".QAct_Speed;
   END_IF;
END_REGION

REGION Network 150: T-51.00 Comm to Blend
   RUNG wire#powerrail
      Contact( "AlwaysTRUE" )
      wire#w1
      Contact( "T-51_HW".State.Tank_Available )
      Coil( "Preparation to Blend"."T-51_HW".Tank_Available )
   END_RUNG
   RUNG wire#w1
      Contact( "T-51_HW".State.Ready_For_Transfer )
      Coil( "Preparation to Blend"."T-51_HW".Product_Ready )
   END_RUNG
   RUNG wire#w1
      Contact( "T-51_HW".IN_FBAV_Outlet )
      Contact( "T-51_HW".IN_FBAV_Transfer )
      Coil( "Preparation to Blend"."T-51_HW".Valve_Open )
   END_RUNG
   RUNG wire#w1
      Contact( "T-51_HW".IN_FBP_Transfer )
      Coil( "Preparation to Blend"."T-51_HW".Pump_Run )
   END_RUNG
   // the same network as SCL:
   "Preparation to Blend"."T-51_HW".Tank_Available := "AlwaysTRUE" AND "T-51_HW".State.Tank_Available;
   "Preparation to Blend"."T-51_HW".Product_Ready := "AlwaysTRUE" AND "T-51_HW".State.Ready_For_Transfer;
   "Preparation to Blend"."T-51_HW".Valve_Open := "AlwaysTRUE" AND "T-51_HW".IN_FBAV_Outlet AND "T-51_HW".IN_FBAV_Transfer;
   "Preparation to Blend"."T-51_HW".Pump_Run := "AlwaysTRUE" AND "T-51_HW".IN_FBP_Transfer;
END_REGION

REGION Network 153: CIP Header 1 and Header 2 Enable
   RUNG wire#powerrail
      Contact( "AlwaysTRUE" )
      I_Contact( "T-02_ChiliAwetan_1".Out_CIP_Req )
      I_Contact( "T-03_ChiliAwetan_2".Out_CIP_Req )
      I_Contact( "T-04_ChiliAwetan_3".Out_CIP_Req )
      I_Contact( "T-09_Garlic".Out_CIP_Req )
      I_Contact( "T-10_Vinegar".Out_CIP_Req )
      I_Contact( "Osa to CIP"."CIP OSA on Process" )
      wire#w1
      I_Contact( "Blend to Preparation"."T-20".LineHeader1_OK )
      I_Contact( "Blend to Preparation"."T-21".LineHeader1_OK )
      I_Contact( "Blend to Preparation"."T-30".LineHeader1_OK )
      I_Contact( "Blend to Preparation"."T-31".LineHeader1_OK )
      I_Contact( "Blend to Preparation"."T-40".LineHeader1_OK )
      I_Contact( "Blend to Preparation"."T-41".LineHeader1_OK )
      Coil( "General Preparation"."Header 1"."CIP Enable" )
   END_RUNG
   RUNG wire#w1
      I_Contact( "Blend to Preparation"."T-20".LineHeader2_OK )
      I_Contact( "Blend to Preparation"."T-21".LineHeader2_OK )
      I_Contact( "Blend to Preparation"."T-30".LineHeader2_OK )
      I_Contact( "Blend to Preparation"."T-31".LineHeader2_OK )
      I_Contact( "Blend to Preparation"."T-40".LineHeader2_OK )
      I_Contact( "Blend to Preparation"."T-41".LineHeader2_OK )
      Coil( "General Preparation"."Header 2"."CIP Enable" )
   END_RUNG
   // the same network as SCL:
   #_w1 := "AlwaysTRUE" AND NOT "T-02_ChiliAwetan_1".Out_CIP_Req AND NOT "T-03_ChiliAwetan_2".Out_CIP_Req AND NOT "T-04_ChiliAwetan_3".Out_CIP_Req AND NOT "T-09_Garlic".Out_CIP_Req AND NOT "T-10_Vinegar".Out_CIP_Req AND NOT "Osa to CIP"."CIP OSA on Process";
   "General Preparation"."Header 1"."CIP Enable" := #_w1 AND NOT "Blend to Preparation"."T-20".LineHeader1_OK AND NOT "Blend to Preparation"."T-21".LineHeader1_OK AND NOT "Blend to Preparation"."T-30".LineHeader1_OK AND NOT "Blend to Preparation"."T-31".LineHeader1_OK AND NOT "Blend to Preparation"."T-40".LineHeader1_OK AND NOT "Blend to Preparation"."T-41".LineHeader1_OK;
   "General Preparation"."Header 2"."CIP Enable" := #_w1 AND NOT "Blend to Preparation"."T-20".LineHeader2_OK AND NOT "Blend to Preparation"."T-21".LineHeader2_OK AND NOT "Blend to Preparation"."T-30".LineHeader2_OK AND NOT "Blend to Preparation"."T-31".LineHeader2_OK AND NOT "Blend to Preparation"."T-40".LineHeader2_OK AND NOT "Blend to Preparation"."T-41".LineHeader2_OK;
END_REGION

REGION Network 154: CIP Header 1 and Header 2 Request
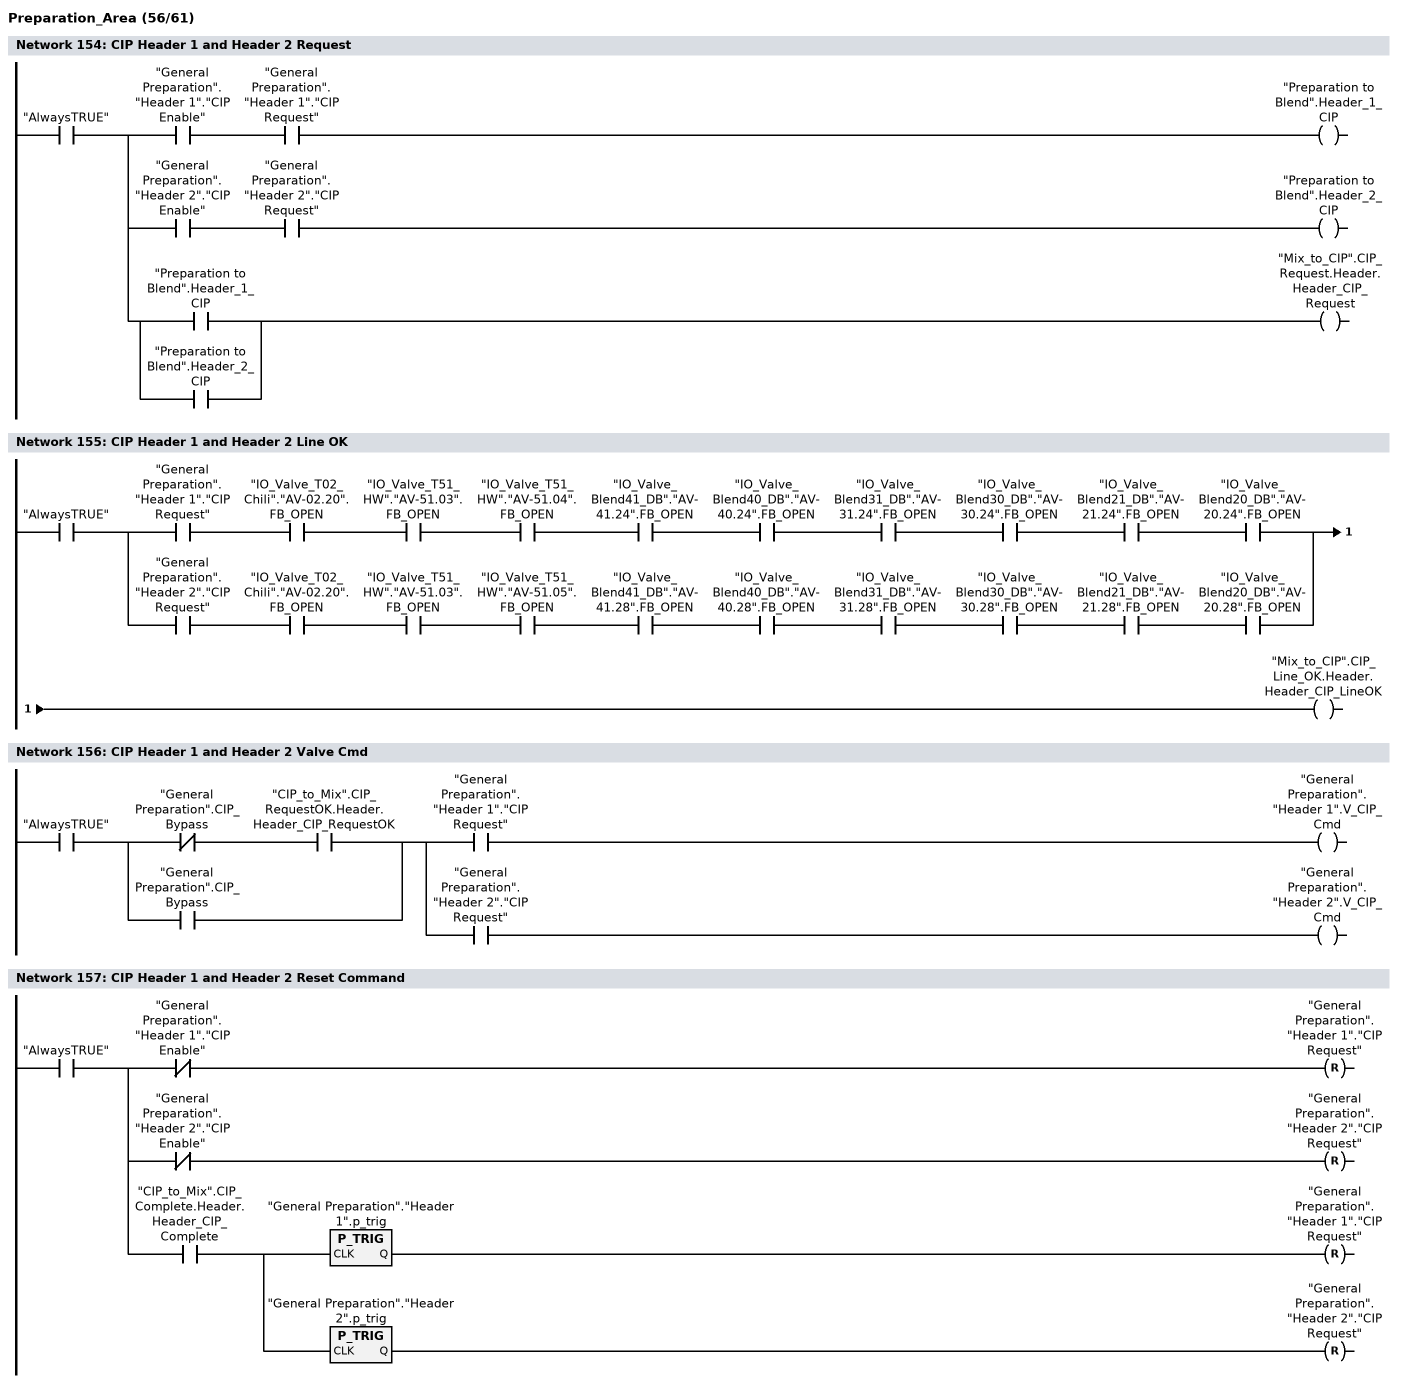
   RUNG wire#powerrail
      Contact( "AlwaysTRUE" )
      wire#w1
      Contact( "General Preparation"."Header 1"."CIP Enable" )
      Contact( "General Preparation"."Header 1"."CIP Request" )
      Coil( "Preparation to Blend".Header_1_CIP )
   END_RUNG
   RUNG wire#w1
      Contact( "General Preparation"."Header 2"."CIP Enable" )
      Contact( "General Preparation"."Header 2"."CIP Request" )
      Coil( "Preparation to Blend".Header_2_CIP )
   END_RUNG
   RUNG wire#w1
      Contact( "Preparation to Blend".Header_1_CIP )
      wire#w2
      Coil( "Mix_to_CIP".CIP_Request.Header.Header_CIP_Request )
   END_RUNG
   RUNG wire#w1
      Contact( "Preparation to Blend".Header_2_CIP )
   END_RUNG wire#w2
   // the same network as SCL:
   "Preparation to Blend".Header_1_CIP := "AlwaysTRUE" AND "General Preparation"."Header 1"."CIP Enable" AND "General Preparation"."Header 1"."CIP Request";
   "Preparation to Blend".Header_2_CIP := "AlwaysTRUE" AND "General Preparation"."Header 2"."CIP Enable" AND "General Preparation"."Header 2"."CIP Request";
   "Mix_to_CIP".CIP_Request.Header.Header_CIP_Request := "AlwaysTRUE" AND ("Preparation to Blend".Header_1_CIP OR "Preparation to Blend".Header_2_CIP);
END_REGION

REGION Network 155: CIP Header 1 and Header 2 Line OK
   RUNG wire#powerrail
      Contact( "AlwaysTRUE" )
      wire#w1
      Contact( "General Preparation"."Header 1"."CIP Request" )
      Contact( "IO_Valve_T02_Chili"."AV-02.20".FB_OPEN )
      Contact( "IO_Valve_T51_HW"."AV-51.03".FB_OPEN )
      Contact( "IO_Valve_T51_HW"."AV-51.04".FB_OPEN )
      Contact( "IO_Valve_Blend41_DB"."AV-41.24".FB_OPEN )
      Contact( "IO_Valve_Blend40_DB"."AV-40.24".FB_OPEN )
      Contact( "IO_Valve_Blend31_DB"."AV-31.24".FB_OPEN )
      Contact( "IO_Valve_Blend30_DB"."AV-30.24".FB_OPEN )
      Contact( "IO_Valve_Blend21_DB"."AV-21.24".FB_OPEN )
      Contact( "IO_Valve_Blend20_DB"."AV-20.24".FB_OPEN )
      wire#w2
      Coil( "Mix_to_CIP".CIP_Line_OK.Header.Header_CIP_LineOK )
   END_RUNG
   RUNG wire#w1
      Contact( "General Preparation"."Header 2"."CIP Request" )
      Contact( "IO_Valve_T02_Chili"."AV-02.20".FB_OPEN )
      Contact( "IO_Valve_T51_HW"."AV-51.03".FB_OPEN )
      Contact( "IO_Valve_T51_HW"."AV-51.05".FB_OPEN )
      Contact( "IO_Valve_Blend41_DB"."AV-41.28".FB_OPEN )
      Contact( "IO_Valve_Blend40_DB"."AV-40.28".FB_OPEN )
      Contact( "IO_Valve_Blend31_DB"."AV-31.28".FB_OPEN )
      Contact( "IO_Valve_Blend30_DB"."AV-30.28".FB_OPEN )
      Contact( "IO_Valve_Blend21_DB"."AV-21.28".FB_OPEN )
      Contact( "IO_Valve_Blend20_DB"."AV-20.28".FB_OPEN )
   END_RUNG wire#w2
   // the same network as SCL:
   "Mix_to_CIP".CIP_Line_OK.Header.Header_CIP_LineOK := "AlwaysTRUE" AND (("General Preparation"."Header 1"."CIP Request" AND "IO_Valve_T02_Chili"."AV-02.20".FB_OPEN AND "IO_Valve_T51_HW"."AV-51.03".FB_OPEN AND "IO_Valve_T51_HW"."AV-51.04".FB_OPEN AND "IO_Valve_Blend41_DB"."AV-41.24".FB_OPEN AND "IO_Valve_Blend40_DB"."AV-40.24".FB_OPEN AND "IO_Valve_Blend31_DB"."AV-31.24".FB_OPEN AND "IO_Valve_Blend30_DB"."AV-30.24".FB_OPEN AND "IO_Valve_Blend21_DB"."AV-21.24".FB_OPEN AND "IO_Valve_Blend20_DB"."AV-20.24".FB_OPEN) OR ("General Preparation"."Header 2"."CIP Request" AND "IO_Valve_T02_Chili"."AV-02.20".FB_OPEN AND "IO_Valve_T51_HW"."AV-51.03".FB_OPEN AND "IO_Valve_T51_HW"."AV-51.05".FB_OPEN AND "IO_Valve_Blend41_DB"."AV-41.28".FB_OPEN AND "IO_Valve_Blend40_DB"."AV-40.28".FB_OPEN AND "IO_Valve_Blend31_DB"."AV-31.28".FB_OPEN AND "IO_Valve_Blend30_DB"."AV-30.28".FB_OPEN AND "IO_Valve_Blend21_DB"."AV-21.28".FB_OPEN AND "IO_Valve_Blend20_DB"."AV-20.28".FB_OPEN));
END_REGION

REGION Network 156: CIP Header 1 and Header 2 Valve Cmd
   RUNG wire#powerrail
      Contact( "AlwaysTRUE" )
      wire#w1
      I_Contact( "General Preparation".CIP_Bypass )
      Contact( "CIP_to_Mix".CIP_RequestOK.Header.Header_CIP_RequestOK )
      wire#w2
      Contact( "General Preparation"."Header 1"."CIP Request" )
      Coil( "General Preparation"."Header 1".V_CIP_Cmd )
   END_RUNG
   RUNG wire#w1
      Contact( "General Preparation".CIP_Bypass )
   END_RUNG wire#w2
   RUNG wire#w2
      Contact( "General Preparation"."Header 2"."CIP Request" )
      Coil( "General Preparation"."Header 2".V_CIP_Cmd )
   END_RUNG
   // the same network as SCL:
   #_w1 := "AlwaysTRUE" AND ((NOT "General Preparation".CIP_Bypass AND "CIP_to_Mix".CIP_RequestOK.Header.Header_CIP_RequestOK) OR "General Preparation".CIP_Bypass);
   "General Preparation"."Header 1".V_CIP_Cmd := #_w1 AND "General Preparation"."Header 1"."CIP Request";
   "General Preparation"."Header 2".V_CIP_Cmd := #_w1 AND "General Preparation"."Header 2"."CIP Request";
END_REGION

REGION Network 157: CIP Header 1 and Header 2 Reset Command
   RUNG wire#powerrail
      Contact( "AlwaysTRUE" )
      wire#w1
      I_Contact( "General Preparation"."Header 1"."CIP Enable" )
      R_Coil( "General Preparation"."Header 1"."CIP Request" )
   END_RUNG
   RUNG wire#w1
      I_Contact( "General Preparation"."Header 2"."CIP Enable" )
      R_Coil( "General Preparation"."Header 2"."CIP Request" )
   END_RUNG
   RUNG wire#w1
      Contact( "CIP_to_Mix".CIP_Complete.Header.Header_CIP_Complete )
      wire#w2
      P_Trig( "General Preparation"."Header 1".p_trig )
      R_Coil( "General Preparation"."Header 1"."CIP Request" )
   END_RUNG
   RUNG wire#w2
      P_Trig( "General Preparation"."Header 2".p_trig )
      R_Coil( "General Preparation"."Header 2"."CIP Request" )
   END_RUNG
   // the same network as SCL:
   IF "AlwaysTRUE" AND NOT "General Preparation"."Header 1"."CIP Enable" THEN
       "General Preparation"."Header 1"."CIP Request" := FALSE;
   END_IF;
   IF "AlwaysTRUE" AND NOT "General Preparation"."Header 2"."CIP Enable" THEN
       "General Preparation"."Header 2"."CIP Request" := FALSE;
   END_IF;
   #_w1 := "AlwaysTRUE" AND "CIP_to_Mix".CIP_Complete.Header.Header_CIP_Complete;
   #_w2 := #_w1 AND NOT "General Preparation"."Header 1".p_trig;   // rising edge
   "General Preparation"."Header 1".p_trig := #_w1;
   IF #_w2 THEN "General Preparation"."Header 1"."CIP Request" := FALSE; END_IF;
   #_w3 := #_w1 AND NOT "General Preparation"."Header 2".p_trig;   // rising edge
   "General Preparation"."Header 2".p_trig := #_w1;
   IF #_w3 THEN "General Preparation"."Header 2"."CIP Request" := FALSE; END_IF;
END_REGION

REGION Network 159: CIP Supply Valve Header 1, Header 2, T-02, T-03, T-04, T-09, T-10 Using AV-02.20
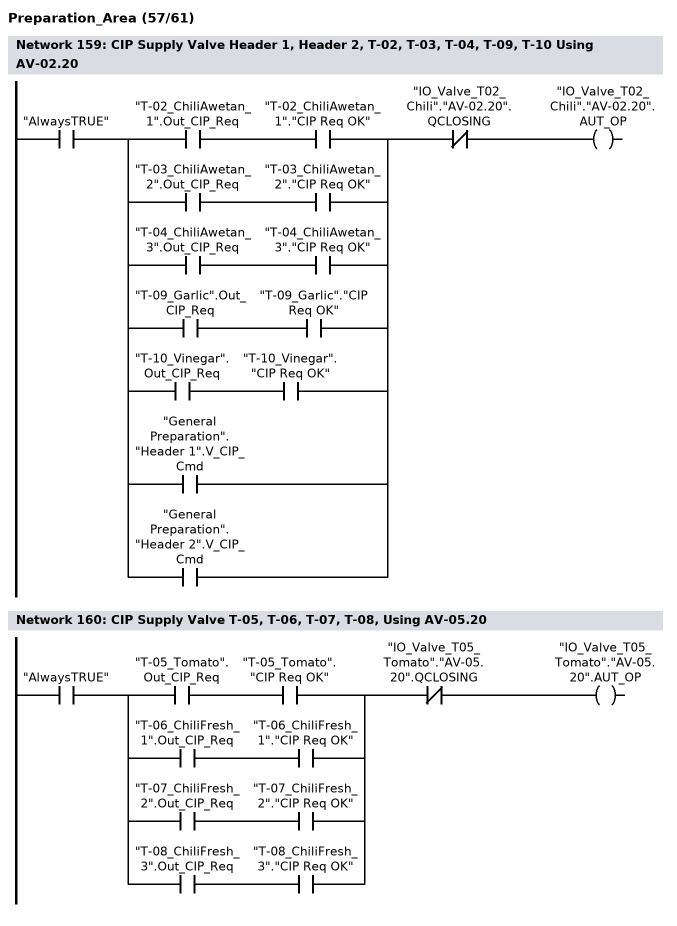
   RUNG wire#powerrail
      Contact( "AlwaysTRUE" )
      wire#w1
      Contact( "T-02_ChiliAwetan_1".Out_CIP_Req )
      Contact( "T-02_ChiliAwetan_1"."CIP Req OK" )
      wire#w2
      I_Contact( "IO_Valve_T02_Chili"."AV-02.20".QCLOSING )
      Coil( "IO_Valve_T02_Chili"."AV-02.20".AUT_OP )
   END_RUNG
   RUNG wire#w1
      Contact( "T-03_ChiliAwetan_2".Out_CIP_Req )
      Contact( "T-03_ChiliAwetan_2"."CIP Req OK" )
   END_RUNG wire#w2
   RUNG wire#w1
      Contact( "T-04_ChiliAwetan_3".Out_CIP_Req )
      Contact( "T-04_ChiliAwetan_3"."CIP Req OK" )
   END_RUNG wire#w2
   RUNG wire#w1
      Contact( "T-09_Garlic".Out_CIP_Req )
      Contact( "T-09_Garlic"."CIP Req OK" )
   END_RUNG wire#w2
   RUNG wire#w1
      Contact( "T-10_Vinegar".Out_CIP_Req )
      Contact( "T-10_Vinegar"."CIP Req OK" )
   END_RUNG wire#w2
   RUNG wire#w1
      Contact( "General Preparation"."Header 1".V_CIP_Cmd )
   END_RUNG wire#w2
   RUNG wire#w1
      Contact( "General Preparation"."Header 2".V_CIP_Cmd )
   END_RUNG wire#w2
   // the same network as SCL:
   "IO_Valve_T02_Chili"."AV-02.20".AUT_OP := "AlwaysTRUE" AND (("T-02_ChiliAwetan_1".Out_CIP_Req AND "T-02_ChiliAwetan_1"."CIP Req OK") OR ("T-03_ChiliAwetan_2".Out_CIP_Req AND "T-03_ChiliAwetan_2"."CIP Req OK") OR ("T-04_ChiliAwetan_3".Out_CIP_Req AND "T-04_ChiliAwetan_3"."CIP Req OK") OR ("T-09_Garlic".Out_CIP_Req AND "T-09_Garlic"."CIP Req OK") OR ("T-10_Vinegar".Out_CIP_Req AND "T-10_Vinegar"."CIP Req OK") OR "General Preparation"."Header 1".V_CIP_Cmd OR "General Preparation"."Header 2".V_CIP_Cmd) AND NOT "IO_Valve_T02_Chili"."AV-02.20".QCLOSING;
END_REGION

REGION Network 160: CIP Supply Valve T-05, T-06, T-07, T-08, Using AV-05.20
   RUNG wire#powerrail
      Contact( "AlwaysTRUE" )
      wire#w1
      Contact( "T-05_Tomato".Out_CIP_Req )
      Contact( "T-05_Tomato"."CIP Req OK" )
      wire#w2
      I_Contact( "IO_Valve_T05_Tomato"."AV-05.20".QCLOSING )
      Coil( "IO_Valve_T05_Tomato"."AV-05.20".AUT_OP )
   END_RUNG
   RUNG wire#w1
      Contact( "T-06_ChiliFresh_1".Out_CIP_Req )
      Contact( "T-06_ChiliFresh_1"."CIP Req OK" )
   END_RUNG wire#w2
   RUNG wire#w1
      Contact( "T-07_ChiliFresh_2".Out_CIP_Req )
      Contact( "T-07_ChiliFresh_2"."CIP Req OK" )
   END_RUNG wire#w2
   RUNG wire#w1
      Contact( "T-08_ChiliFresh_3".Out_CIP_Req )
      Contact( "T-08_ChiliFresh_3"."CIP Req OK" )
   END_RUNG wire#w2
   // the same network as SCL:
   "IO_Valve_T05_Tomato"."AV-05.20".AUT_OP := "AlwaysTRUE" AND (("T-05_Tomato".Out_CIP_Req AND "T-05_Tomato"."CIP Req OK") OR ("T-06_ChiliFresh_1".Out_CIP_Req AND "T-06_ChiliFresh_1"."CIP Req OK") OR ("T-07_ChiliFresh_2".Out_CIP_Req AND "T-07_ChiliFresh_2"."CIP Req OK") OR ("T-08_ChiliFresh_3".Out_CIP_Req AND "T-08_ChiliFresh_3"."CIP Req OK")) AND NOT "IO_Valve_T05_Tomato"."AV-05.20".QCLOSING;
END_REGION

REGION Network 162: CIP Return Valve T-02, T-03, T-04, T-09 to CIP R Pump Using AV-08.17
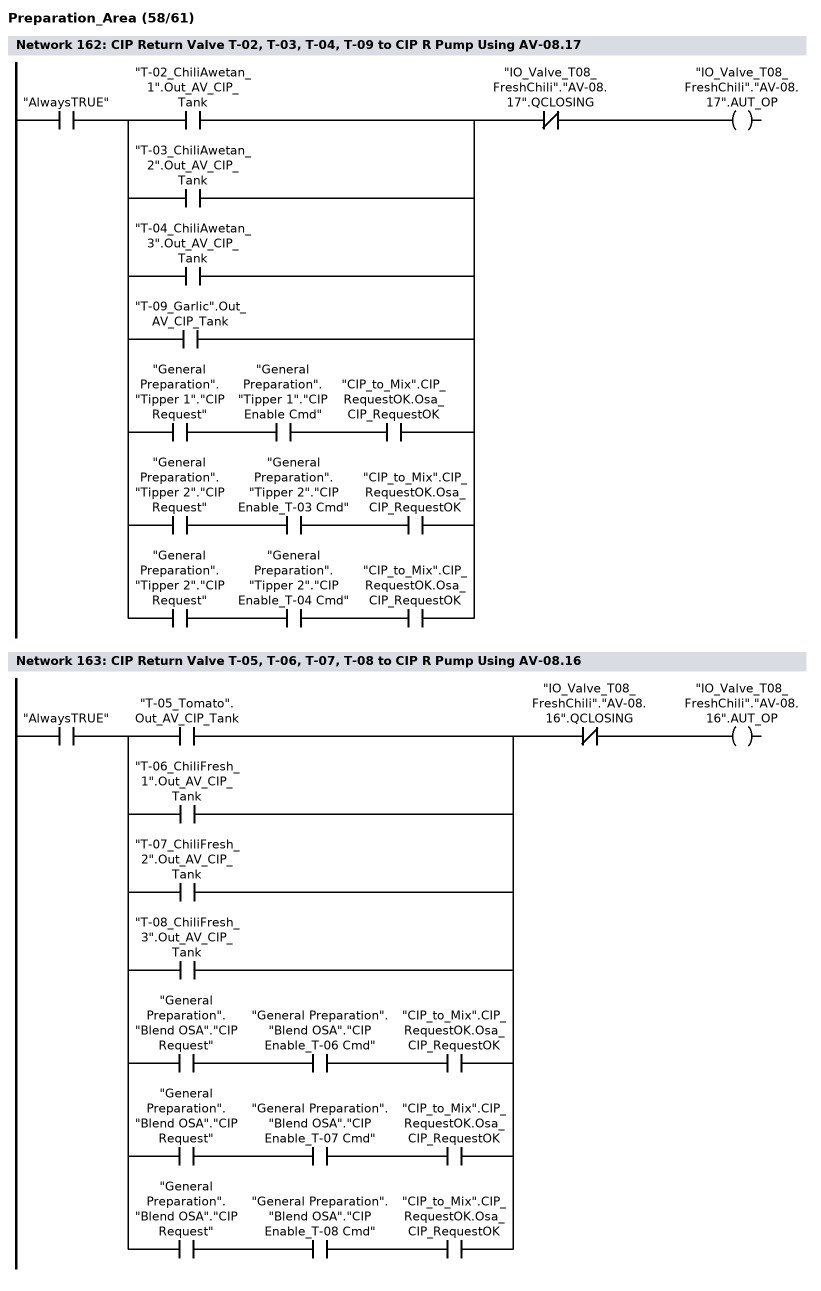
   RUNG wire#powerrail
      Contact( "AlwaysTRUE" )
      wire#w1
      Contact( "T-02_ChiliAwetan_1".Out_AV_CIP_Tank )
      wire#w2
      I_Contact( "IO_Valve_T08_FreshChili"."AV-08.17".QCLOSING )
      Coil( "IO_Valve_T08_FreshChili"."AV-08.17".AUT_OP )
   END_RUNG
   RUNG wire#w1
      Contact( "T-03_ChiliAwetan_2".Out_AV_CIP_Tank )
   END_RUNG wire#w2
   RUNG wire#w1
      Contact( "T-04_ChiliAwetan_3".Out_AV_CIP_Tank )
   END_RUNG wire#w2
   RUNG wire#w1
      Contact( "T-09_Garlic".Out_AV_CIP_Tank )
   END_RUNG wire#w2
   RUNG wire#w1
      Contact( "General Preparation"."Tipper 1"."CIP Request" )
      Contact( "General Preparation"."Tipper 1"."CIP Enable Cmd" )
      Contact( "CIP_to_Mix".CIP_RequestOK.Osa_CIP_RequestOK )
   END_RUNG wire#w2
   RUNG wire#w1
      Contact( "General Preparation"."Tipper 2"."CIP Request" )
      Contact( "General Preparation"."Tipper 2"."CIP Enable_T-03 Cmd" )
      Contact( "CIP_to_Mix".CIP_RequestOK.Osa_CIP_RequestOK )
   END_RUNG wire#w2
   RUNG wire#w1
      Contact( "General Preparation"."Tipper 2"."CIP Request" )
      Contact( "General Preparation"."Tipper 2"."CIP Enable_T-04 Cmd" )
      Contact( "CIP_to_Mix".CIP_RequestOK.Osa_CIP_RequestOK )
   END_RUNG wire#w2
   // the same network as SCL:
   "IO_Valve_T08_FreshChili"."AV-08.17".AUT_OP := "AlwaysTRUE" AND ("T-02_ChiliAwetan_1".Out_AV_CIP_Tank OR "T-03_ChiliAwetan_2".Out_AV_CIP_Tank OR "T-04_ChiliAwetan_3".Out_AV_CIP_Tank OR "T-09_Garlic".Out_AV_CIP_Tank OR ("General Preparation"."Tipper 1"."CIP Request" AND "General Preparation"."Tipper 1"."CIP Enable Cmd" AND "CIP_to_Mix".CIP_RequestOK.Osa_CIP_RequestOK) OR ("General Preparation"."Tipper 2"."CIP Request" AND "General Preparation"."Tipper 2"."CIP Enable_T-03 Cmd" AND "CIP_to_Mix".CIP_RequestOK.Osa_CIP_RequestOK) OR ("General Preparation"."Tipper 2"."CIP Request" AND "General Preparation"."Tipper 2"."CIP Enable_T-04 Cmd" AND "CIP_to_Mix".CIP_RequestOK.Osa_CIP_RequestOK)) AND NOT "IO_Valve_T08_FreshChili"."AV-08.17".QCLOSING;
END_REGION

REGION Network 163: CIP Return Valve T-05, T-06, T-07, T-08 to CIP R Pump Using AV-08.16
   RUNG wire#powerrail
      Contact( "AlwaysTRUE" )
      wire#w1
      Contact( "T-05_Tomato".Out_AV_CIP_Tank )
      wire#w2
      I_Contact( "IO_Valve_T08_FreshChili"."AV-08.16".QCLOSING )
      Coil( "IO_Valve_T08_FreshChili"."AV-08.16".AUT_OP )
   END_RUNG
   RUNG wire#w1
      Contact( "T-06_ChiliFresh_1".Out_AV_CIP_Tank )
   END_RUNG wire#w2
   RUNG wire#w1
      Contact( "T-07_ChiliFresh_2".Out_AV_CIP_Tank )
   END_RUNG wire#w2
   RUNG wire#w1
      Contact( "T-08_ChiliFresh_3".Out_AV_CIP_Tank )
   END_RUNG wire#w2
   RUNG wire#w1
      Contact( "General Preparation"."Blend OSA"."CIP Request" )
      Contact( "General Preparation"."Blend OSA"."CIP Enable_T-06 Cmd" )
      Contact( "CIP_to_Mix".CIP_RequestOK.Osa_CIP_RequestOK )
   END_RUNG wire#w2
   RUNG wire#w1
      Contact( "General Preparation"."Blend OSA"."CIP Request" )
      Contact( "General Preparation"."Blend OSA"."CIP Enable_T-07 Cmd" )
      Contact( "CIP_to_Mix".CIP_RequestOK.Osa_CIP_RequestOK )
   END_RUNG wire#w2
   RUNG wire#w1
      Contact( "General Preparation"."Blend OSA"."CIP Request" )
      Contact( "General Preparation"."Blend OSA"."CIP Enable_T-08 Cmd" )
      Contact( "CIP_to_Mix".CIP_RequestOK.Osa_CIP_RequestOK )
   END_RUNG wire#w2
   // the same network as SCL:
   "IO_Valve_T08_FreshChili"."AV-08.16".AUT_OP := "AlwaysTRUE" AND ("T-05_Tomato".Out_AV_CIP_Tank OR "T-06_ChiliFresh_1".Out_AV_CIP_Tank OR "T-07_ChiliFresh_2".Out_AV_CIP_Tank OR "T-08_ChiliFresh_3".Out_AV_CIP_Tank OR ("General Preparation"."Blend OSA"."CIP Request" AND "General Preparation"."Blend OSA"."CIP Enable_T-06 Cmd" AND "CIP_to_Mix".CIP_RequestOK.Osa_CIP_RequestOK) OR ("General Preparation"."Blend OSA"."CIP Request" AND "General Preparation"."Blend OSA"."CIP Enable_T-07 Cmd" AND "CIP_to_Mix".CIP_RequestOK.Osa_CIP_RequestOK) OR ("General Preparation"."Blend OSA"."CIP Request" AND "General Preparation"."Blend OSA"."CIP Enable_T-08 Cmd" AND "CIP_to_Mix".CIP_RequestOK.Osa_CIP_RequestOK)) AND NOT "IO_Valve_T08_FreshChili"."AV-08.16".QCLOSING;
END_REGION

REGION Network 165: CIP Return Drain Valve T-02, T-03, T-04, T-09 Using AV-02.06
END_REGION

REGION Network 166: CIP Return Drain Valve T-05, T-06, T-07, T-08 Using AV-05.14
END_REGION

REGION Network 168: Drain Valve Flushing AV-08.14 & AV-08.15
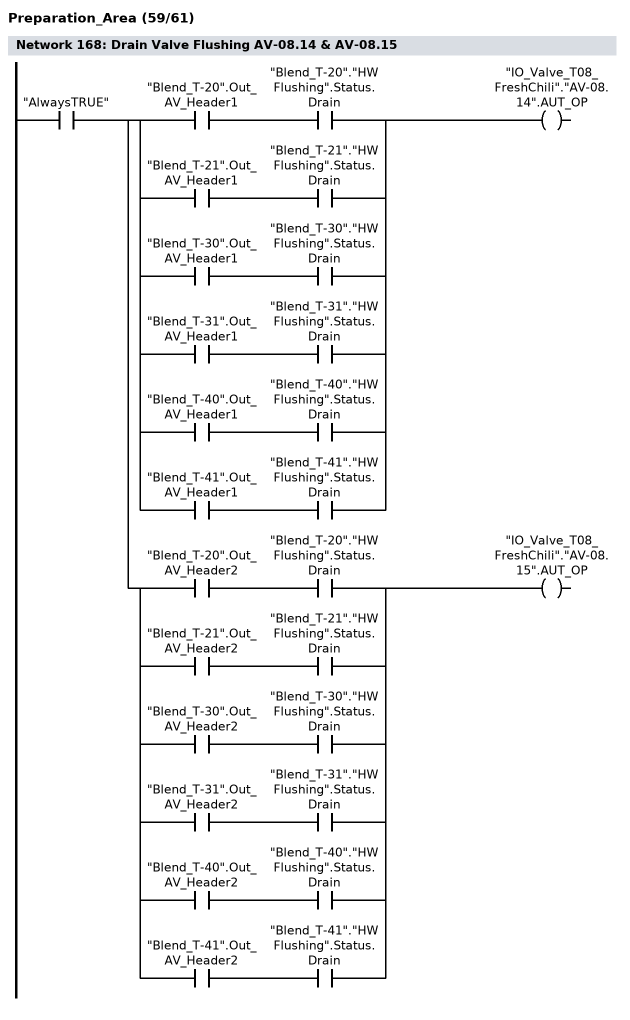
   RUNG wire#powerrail
      Contact( "AlwaysTRUE" )
      wire#w1
      Contact( "Blend_T-20".Out_AV_Header1 )
      Contact( "Blend_T-20"."HW Flushing".Status.Drain )
      wire#w2
      Coil( "IO_Valve_T08_FreshChili"."AV-08.14".AUT_OP )
   END_RUNG
   RUNG wire#w1
      Contact( "Blend_T-21".Out_AV_Header1 )
      Contact( "Blend_T-21"."HW Flushing".Status.Drain )
   END_RUNG wire#w2
   RUNG wire#w1
      Contact( "Blend_T-30".Out_AV_Header1 )
      Contact( "Blend_T-30"."HW Flushing".Status.Drain )
   END_RUNG wire#w2
   RUNG wire#w1
      Contact( "Blend_T-31".Out_AV_Header1 )
      Contact( "Blend_T-31"."HW Flushing".Status.Drain )
   END_RUNG wire#w2
   RUNG wire#w1
      Contact( "Blend_T-40".Out_AV_Header1 )
      Contact( "Blend_T-40"."HW Flushing".Status.Drain )
   END_RUNG wire#w2
   RUNG wire#w1
      Contact( "Blend_T-41".Out_AV_Header1 )
      Contact( "Blend_T-41"."HW Flushing".Status.Drain )
   END_RUNG wire#w2
   RUNG wire#w1
      Contact( "Blend_T-20".Out_AV_Header2 )
      Contact( "Blend_T-20"."HW Flushing".Status.Drain )
      wire#w3
      Coil( "IO_Valve_T08_FreshChili"."AV-08.15".AUT_OP )
   END_RUNG
   RUNG wire#w1
      Contact( "Blend_T-21".Out_AV_Header2 )
      Contact( "Blend_T-21"."HW Flushing".Status.Drain )
   END_RUNG wire#w3
   RUNG wire#w1
      Contact( "Blend_T-30".Out_AV_Header2 )
      Contact( "Blend_T-30"."HW Flushing".Status.Drain )
   END_RUNG wire#w3
   RUNG wire#w1
      Contact( "Blend_T-31".Out_AV_Header2 )
      Contact( "Blend_T-31"."HW Flushing".Status.Drain )
   END_RUNG wire#w3
   RUNG wire#w1
      Contact( "Blend_T-40".Out_AV_Header2 )
      Contact( "Blend_T-40"."HW Flushing".Status.Drain )
   END_RUNG wire#w3
   RUNG wire#w1
      Contact( "Blend_T-41".Out_AV_Header2 )
      Contact( "Blend_T-41"."HW Flushing".Status.Drain )
   END_RUNG wire#w3
   // the same network as SCL:
   "IO_Valve_T08_FreshChili"."AV-08.14".AUT_OP := "AlwaysTRUE" AND (("Blend_T-20".Out_AV_Header1 AND "Blend_T-20"."HW Flushing".Status.Drain) OR ("Blend_T-21".Out_AV_Header1 AND "Blend_T-21"."HW Flushing".Status.Drain) OR ("Blend_T-30".Out_AV_Header1 AND "Blend_T-30"."HW Flushing".Status.Drain) OR ("Blend_T-31".Out_AV_Header1 AND "Blend_T-31"."HW Flushing".Status.Drain) OR ("Blend_T-40".Out_AV_Header1 AND "Blend_T-40"."HW Flushing".Status.Drain) OR ("Blend_T-41".Out_AV_Header1 AND "Blend_T-41"."HW Flushing".Status.Drain));
   "IO_Valve_T08_FreshChili"."AV-08.15".AUT_OP := "AlwaysTRUE" AND (("Blend_T-20".Out_AV_Header2 AND "Blend_T-20"."HW Flushing".Status.Drain) OR ("Blend_T-21".Out_AV_Header2 AND "Blend_T-21"."HW Flushing".Status.Drain) OR ("Blend_T-30".Out_AV_Header2 AND "Blend_T-30"."HW Flushing".Status.Drain) OR ("Blend_T-31".Out_AV_Header2 AND "Blend_T-31"."HW Flushing".Status.Drain) OR ("Blend_T-40".Out_AV_Header2 AND "Blend_T-40"."HW Flushing".Status.Drain) OR ("Blend_T-41".Out_AV_Header2 AND "Blend_T-41"."HW Flushing".Status.Drain));
END_REGION

REGION Network 170: CIP Return Pump Using P-08.02 (Command)
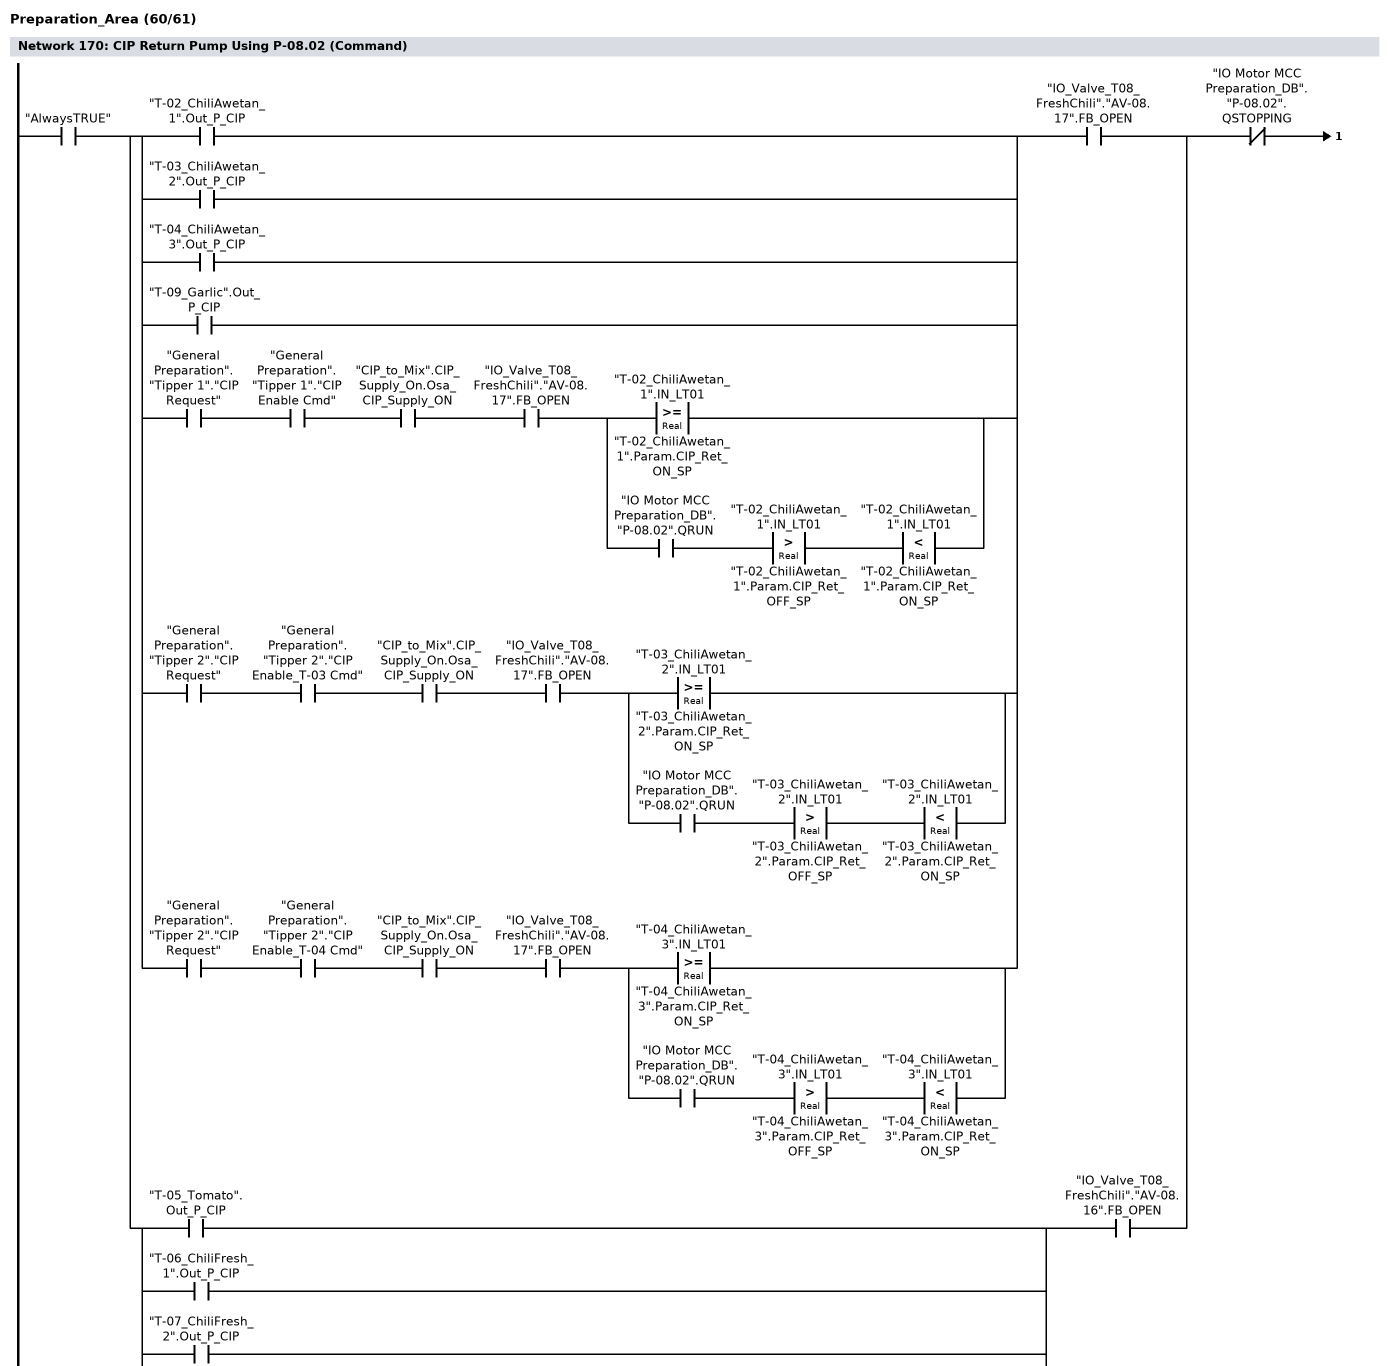
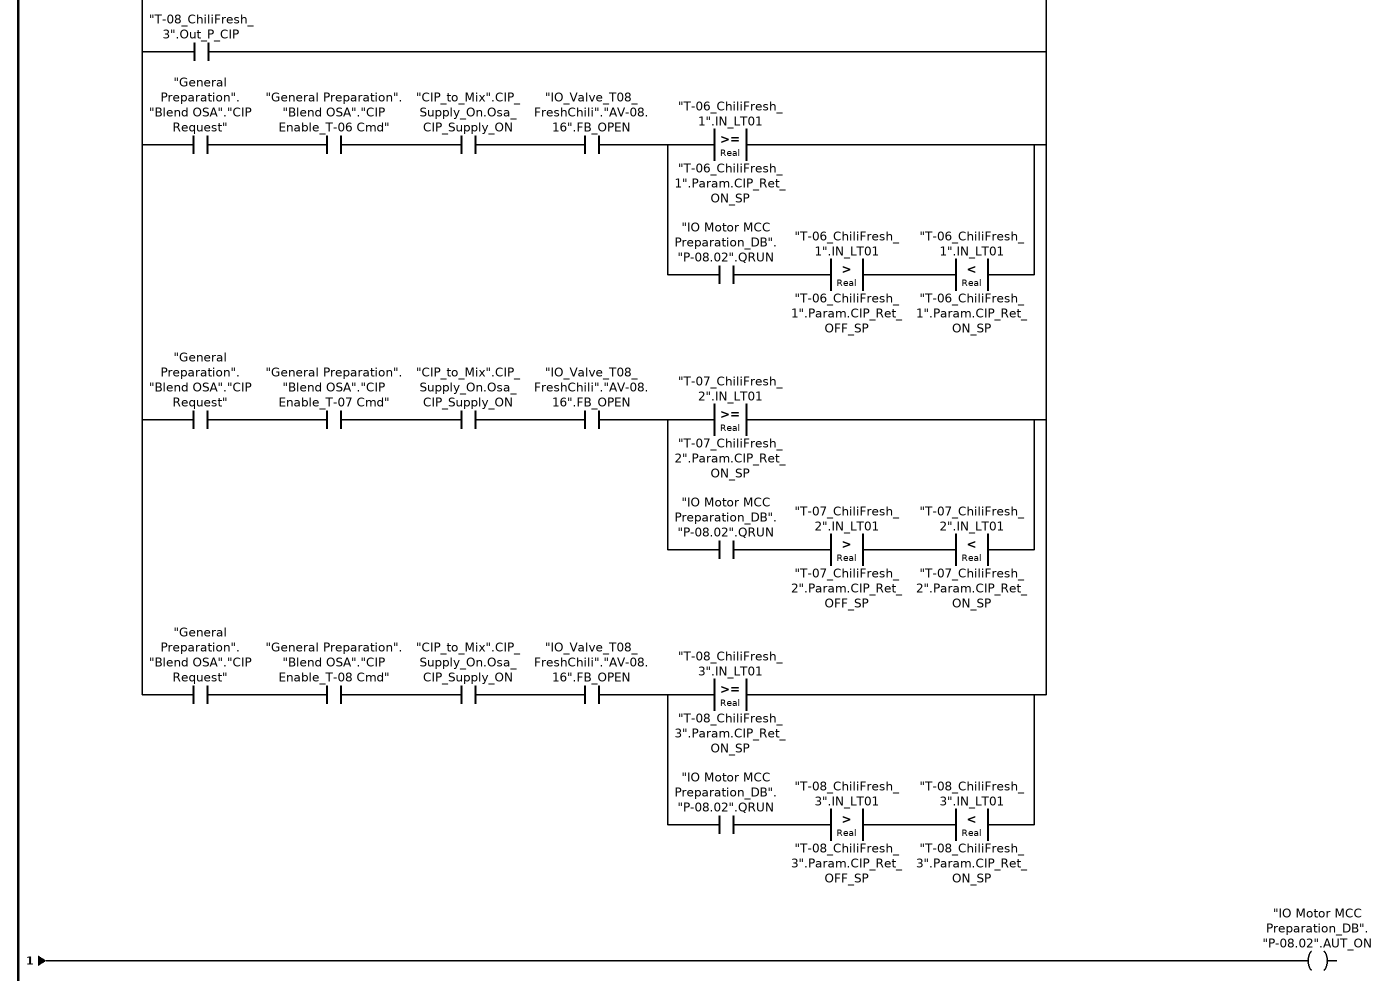
   RUNG wire#powerrail
      Contact( "AlwaysTRUE" )
      wire#w1
      Contact( "T-02_ChiliAwetan_1".Out_P_CIP )
      wire#w2
      Contact( "IO_Valve_T08_FreshChili"."AV-08.17".FB_OPEN )
      wire#w6
      I_Contact( "IO Motor MCC Preparation_DB"."P-08.02".QSTOPPING )
      Coil( "IO Motor MCC Preparation_DB"."P-08.02".AUT_ON )
   END_RUNG
   RUNG wire#w1
      Contact( "T-03_ChiliAwetan_2".Out_P_CIP )
   END_RUNG wire#w2
   RUNG wire#w1
      Contact( "T-04_ChiliAwetan_3".Out_P_CIP )
   END_RUNG wire#w2
   RUNG wire#w1
      Contact( "T-09_Garlic".Out_P_CIP )
   END_RUNG wire#w2
   RUNG wire#w1
      Contact( "General Preparation"."Tipper 1"."CIP Request" )
      Contact( "General Preparation"."Tipper 1"."CIP Enable Cmd" )
      Contact( "CIP_to_Mix".CIP_Supply_On.Osa_CIP_Supply_ON )
      Contact( "IO_Valve_T08_FreshChili"."AV-08.17".FB_OPEN )
      wire#w3
      { S7_Templates := "SrcType := Real" } GE_Contact(in1 := "T-02_ChiliAwetan_1".IN_LT01, in2 := "T-02_ChiliAwetan_1".Param.CIP_Ret_ON_SP)
   END_RUNG wire#w2
   RUNG wire#w3
      Contact( "IO Motor MCC Preparation_DB"."P-08.02".QRUN )
      { S7_Templates := "SrcType := Real" } GT_Contact(in1 := "T-02_ChiliAwetan_1".IN_LT01, in2 := "T-02_ChiliAwetan_1".Param.CIP_Ret_OFF_SP)
      { S7_Templates := "SrcType := Real" } LT_Contact(in1 := "T-02_ChiliAwetan_1".IN_LT01, in2 := "T-02_ChiliAwetan_1".Param.CIP_Ret_ON_SP)
   END_RUNG wire#w2
   RUNG wire#w1
      Contact( "General Preparation"."Tipper 2"."CIP Request" )
      Contact( "General Preparation"."Tipper 2"."CIP Enable_T-03 Cmd" )
      Contact( "CIP_to_Mix".CIP_Supply_On.Osa_CIP_Supply_ON )
      Contact( "IO_Valve_T08_FreshChili"."AV-08.17".FB_OPEN )
      wire#w4
      { S7_Templates := "SrcType := Real" } GE_Contact(in1 := "T-03_ChiliAwetan_2".IN_LT01, in2 := "T-03_ChiliAwetan_2".Param.CIP_Ret_ON_SP)
   END_RUNG wire#w2
   RUNG wire#w4
      Contact( "IO Motor MCC Preparation_DB"."P-08.02".QRUN )
      { S7_Templates := "SrcType := Real" } GT_Contact(in1 := "T-03_ChiliAwetan_2".IN_LT01, in2 := "T-03_ChiliAwetan_2".Param.CIP_Ret_OFF_SP)
      { S7_Templates := "SrcType := Real" } LT_Contact(in1 := "T-03_ChiliAwetan_2".IN_LT01, in2 := "T-03_ChiliAwetan_2".Param.CIP_Ret_ON_SP)
   END_RUNG wire#w2
   RUNG wire#w1
      Contact( "General Preparation"."Tipper 2"."CIP Request" )
      Contact( "General Preparation"."Tipper 2"."CIP Enable_T-04 Cmd" )
      Contact( "CIP_to_Mix".CIP_Supply_On.Osa_CIP_Supply_ON )
      Contact( "IO_Valve_T08_FreshChili"."AV-08.17".FB_OPEN )
      wire#w5
      { S7_Templates := "SrcType := Real" } GE_Contact(in1 := "T-04_ChiliAwetan_3".IN_LT01, in2 := "T-04_ChiliAwetan_3".Param.CIP_Ret_ON_SP)
   END_RUNG wire#w2
   RUNG wire#w5
      Contact( "IO Motor MCC Preparation_DB"."P-08.02".QRUN )
      { S7_Templates := "SrcType := Real" } GT_Contact(in1 := "T-04_ChiliAwetan_3".IN_LT01, in2 := "T-04_ChiliAwetan_3".Param.CIP_Ret_OFF_SP)
      { S7_Templates := "SrcType := Real" } LT_Contact(in1 := "T-04_ChiliAwetan_3".IN_LT01, in2 := "T-04_ChiliAwetan_3".Param.CIP_Ret_ON_SP)
   END_RUNG wire#w2
   RUNG wire#w1
      Contact( "T-05_Tomato".Out_P_CIP )
      wire#w7
      Contact( "IO_Valve_T08_FreshChili"."AV-08.16".FB_OPEN )
   END_RUNG wire#w6
   RUNG wire#w1
      Contact( "T-06_ChiliFresh_1".Out_P_CIP )
   END_RUNG wire#w7
   RUNG wire#w1
      Contact( "T-07_ChiliFresh_2".Out_P_CIP )
   END_RUNG wire#w7
   RUNG wire#w1
      Contact( "T-08_ChiliFresh_3".Out_P_CIP )
   END_RUNG wire#w7
   RUNG wire#w1
      Contact( "General Preparation"."Blend OSA"."CIP Request" )
      Contact( "General Preparation"."Blend OSA"."CIP Enable_T-06 Cmd" )
      Contact( "CIP_to_Mix".CIP_Supply_On.Osa_CIP_Supply_ON )
      Contact( "IO_Valve_T08_FreshChili"."AV-08.16".FB_OPEN )
      wire#w8
      { S7_Templates := "SrcType := Real" } GE_Contact(in1 := "T-06_ChiliFresh_1".IN_LT01, in2 := "T-06_ChiliFresh_1".Param.CIP_Ret_ON_SP)
   END_RUNG wire#w7
   RUNG wire#w8
      Contact( "IO Motor MCC Preparation_DB"."P-08.02".QRUN )
      { S7_Templates := "SrcType := Real" } GT_Contact(in1 := "T-06_ChiliFresh_1".IN_LT01, in2 := "T-06_ChiliFresh_1".Param.CIP_Ret_OFF_SP)
      { S7_Templates := "SrcType := Real" } LT_Contact(in1 := "T-06_ChiliFresh_1".IN_LT01, in2 := "T-06_ChiliFresh_1".Param.CIP_Ret_ON_SP)
   END_RUNG wire#w7
   RUNG wire#w1
      Contact( "General Preparation"."Blend OSA"."CIP Request" )
      Contact( "General Preparation"."Blend OSA"."CIP Enable_T-07 Cmd" )
      Contact( "CIP_to_Mix".CIP_Supply_On.Osa_CIP_Supply_ON )
      Contact( "IO_Valve_T08_FreshChili"."AV-08.16".FB_OPEN )
      wire#w9
      { S7_Templates := "SrcType := Real" } GE_Contact(in1 := "T-07_ChiliFresh_2".IN_LT01, in2 := "T-07_ChiliFresh_2".Param.CIP_Ret_ON_SP)
   END_RUNG wire#w7
   RUNG wire#w9
      Contact( "IO Motor MCC Preparation_DB"."P-08.02".QRUN )
      { S7_Templates := "SrcType := Real" } GT_Contact(in1 := "T-07_ChiliFresh_2".IN_LT01, in2 := "T-07_ChiliFresh_2".Param.CIP_Ret_OFF_SP)
      { S7_Templates := "SrcType := Real" } LT_Contact(in1 := "T-07_ChiliFresh_2".IN_LT01, in2 := "T-07_ChiliFresh_2".Param.CIP_Ret_ON_SP)
   END_RUNG wire#w7
   RUNG wire#w1
      Contact( "General Preparation"."Blend OSA"."CIP Request" )
      Contact( "General Preparation"."Blend OSA"."CIP Enable_T-08 Cmd" )
      Contact( "CIP_to_Mix".CIP_Supply_On.Osa_CIP_Supply_ON )
      Contact( "IO_Valve_T08_FreshChili"."AV-08.16".FB_OPEN )
      wire#w10
      { S7_Templates := "SrcType := Real" } GE_Contact(in1 := "T-08_ChiliFresh_3".IN_LT01, in2 := "T-08_ChiliFresh_3".Param.CIP_Ret_ON_SP)
   END_RUNG wire#w7
   RUNG wire#w10
      Contact( "IO Motor MCC Preparation_DB"."P-08.02".QRUN )
      { S7_Templates := "SrcType := Real" } GT_Contact(in1 := "T-08_ChiliFresh_3".IN_LT01, in2 := "T-08_ChiliFresh_3".Param.CIP_Ret_OFF_SP)
      { S7_Templates := "SrcType := Real" } LT_Contact(in1 := "T-08_ChiliFresh_3".IN_LT01, in2 := "T-08_ChiliFresh_3".Param.CIP_Ret_ON_SP)
   END_RUNG wire#w7
   // the same network as SCL:
   "IO Motor MCC Preparation_DB"."P-08.02".AUT_ON := "AlwaysTRUE" AND ((("T-02_ChiliAwetan_1".Out_P_CIP OR "T-03_ChiliAwetan_2".Out_P_CIP OR "T-04_ChiliAwetan_3".Out_P_CIP OR "T-09_Garlic".Out_P_CIP OR ("General Preparation"."Tipper 1"."CIP Request" AND "General Preparation"."Tipper 1"."CIP Enable Cmd" AND "CIP_to_Mix".CIP_Supply_On.Osa_CIP_Supply_ON AND "IO_Valve_T08_FreshChili"."AV-08.17".FB_OPEN AND (("T-02_ChiliAwetan_1".IN_LT01 >= "T-02_ChiliAwetan_1".Param.CIP_Ret_ON_SP) OR ("IO Motor MCC Preparation_DB"."P-08.02".QRUN AND ("T-02_ChiliAwetan_1".IN_LT01 > "T-02_ChiliAwetan_1".Param.CIP_Ret_OFF_SP) AND ("T-02_ChiliAwetan_1".IN_LT01 < "T-02_ChiliAwetan_1".Param.CIP_Ret_ON_SP)))) OR ("General Preparation"."Tipper 2"."CIP Request" AND "General Preparation"."Tipper 2"."CIP Enable_T-03 Cmd" AND "CIP_to_Mix".CIP_Supply_On.Osa_CIP_Supply_ON AND "IO_Valve_T08_FreshChili"."AV-08.17".FB_OPEN AND (("T-03_ChiliAwetan_2".IN_LT01 >= "T-03_ChiliAwetan_2".Param.CIP_Ret_ON_SP) OR ("IO Motor MCC Preparation_DB"."P-08.02".QRUN AND ("T-03_ChiliAwetan_2".IN_LT01 > "T-03_ChiliAwetan_2".Param.CIP_Ret_OFF_SP) AND ("T-03_ChiliAwetan_2".IN_LT01 < "T-03_ChiliAwetan_2".Param.CIP_Ret_ON_SP)))) OR ("General Preparation"."Tipper 2"."CIP Request" AND "General Preparation"."Tipper 2"."CIP Enable_T-04 Cmd" AND "CIP_to_Mix".CIP_Supply_On.Osa_CIP_Supply_ON AND "IO_Valve_T08_FreshChili"."AV-08.17".FB_OPEN AND (("T-04_ChiliAwetan_3".IN_LT01 >= "T-04_ChiliAwetan_3".Param.CIP_Ret_ON_SP) OR ("IO Motor MCC Preparation_DB"."P-08.02".QRUN AND ("T-04_ChiliAwetan_3".IN_LT01 > "T-04_ChiliAwetan_3".Param.CIP_Ret_OFF_SP) AND ("T-04_ChiliAwetan_3".IN_LT01 < "T-04_ChiliAwetan_3".Param.CIP_Ret_ON_SP))))) AND "IO_Valve_T08_FreshChili"."AV-08.17".FB_OPEN) OR (("T-05_Tomato".Out_P_CIP OR "T-06_ChiliFresh_1".Out_P_CIP OR "T-07_ChiliFresh_2".Out_P_CIP OR "T-08_ChiliFresh_3".Out_P_CIP OR ("General Preparation"."Blend OSA"."CIP Request" AND "General Preparation"."Blend OSA"."CIP Enable_T-06 Cmd" AND "CIP_to_Mix".CIP_Supply_On.Osa_CIP_Supply_ON AND "IO_Valve_T08_FreshChili"."AV-08.16".FB_OPEN AND (("T-06_ChiliFresh_1".IN_LT01 >= "T-06_ChiliFresh_1".Param.CIP_Ret_ON_SP) OR ("IO Motor MCC Preparation_DB"."P-08.02".QRUN AND ("T-06_ChiliFresh_1".IN_LT01 > "T-06_ChiliFresh_1".Param.CIP_Ret_OFF_SP) AND ("T-06_ChiliFresh_1".IN_LT01 < "T-06_ChiliFresh_1".Param.CIP_Ret_ON_SP)))) OR ("General Preparation"."Blend OSA"."CIP Request" AND "General Preparation"."Blend OSA"."CIP Enable_T-07 Cmd" AND "CIP_to_Mix".CIP_Supply_On.Osa_CIP_Supply_ON AND "IO_Valve_T08_FreshChili"."AV-08.16".FB_OPEN AND (("T-07_ChiliFresh_2".IN_LT01 >= "T-07_ChiliFresh_2".Param.CIP_Ret_ON_SP) OR ("IO Motor MCC Preparation_DB"."P-08.02".QRUN AND ("T-07_ChiliFresh_2".IN_LT01 > "T-07_ChiliFresh_2".Param.CIP_Ret_OFF_SP) AND ("T-07_ChiliFresh_2".IN_LT01 < "T-07_ChiliFresh_2".Param.CIP_Ret_ON_SP)))) OR ("General Preparation"."Blend OSA"."CIP Request" AND "General Preparation"."Blend OSA"."CIP Enable_T-08 Cmd" AND "CIP_to_Mix".CIP_Supply_On.Osa_CIP_Supply_ON AND "IO_Valve_T08_FreshChili"."AV-08.16".FB_OPEN AND (("T-08_ChiliFresh_3".IN_LT01 >= "T-08_ChiliFresh_3".Param.CIP_Ret_ON_SP) OR ("IO Motor MCC Preparation_DB"."P-08.02".QRUN AND ("T-08_ChiliFresh_3".IN_LT01 > "T-08_ChiliFresh_3".Param.CIP_Ret_OFF_SP) AND ("T-08_ChiliFresh_3".IN_LT01 < "T-08_ChiliFresh_3".Param.CIP_Ret_ON_SP))))) AND "IO_Valve_T08_FreshChili"."AV-08.16".FB_OPEN)) AND NOT "IO Motor MCC Preparation_DB"."P-08.02".QSTOPPING;
END_REGION

REGION Network 171: CIP Return Pump Using P-08.02 (Speed)
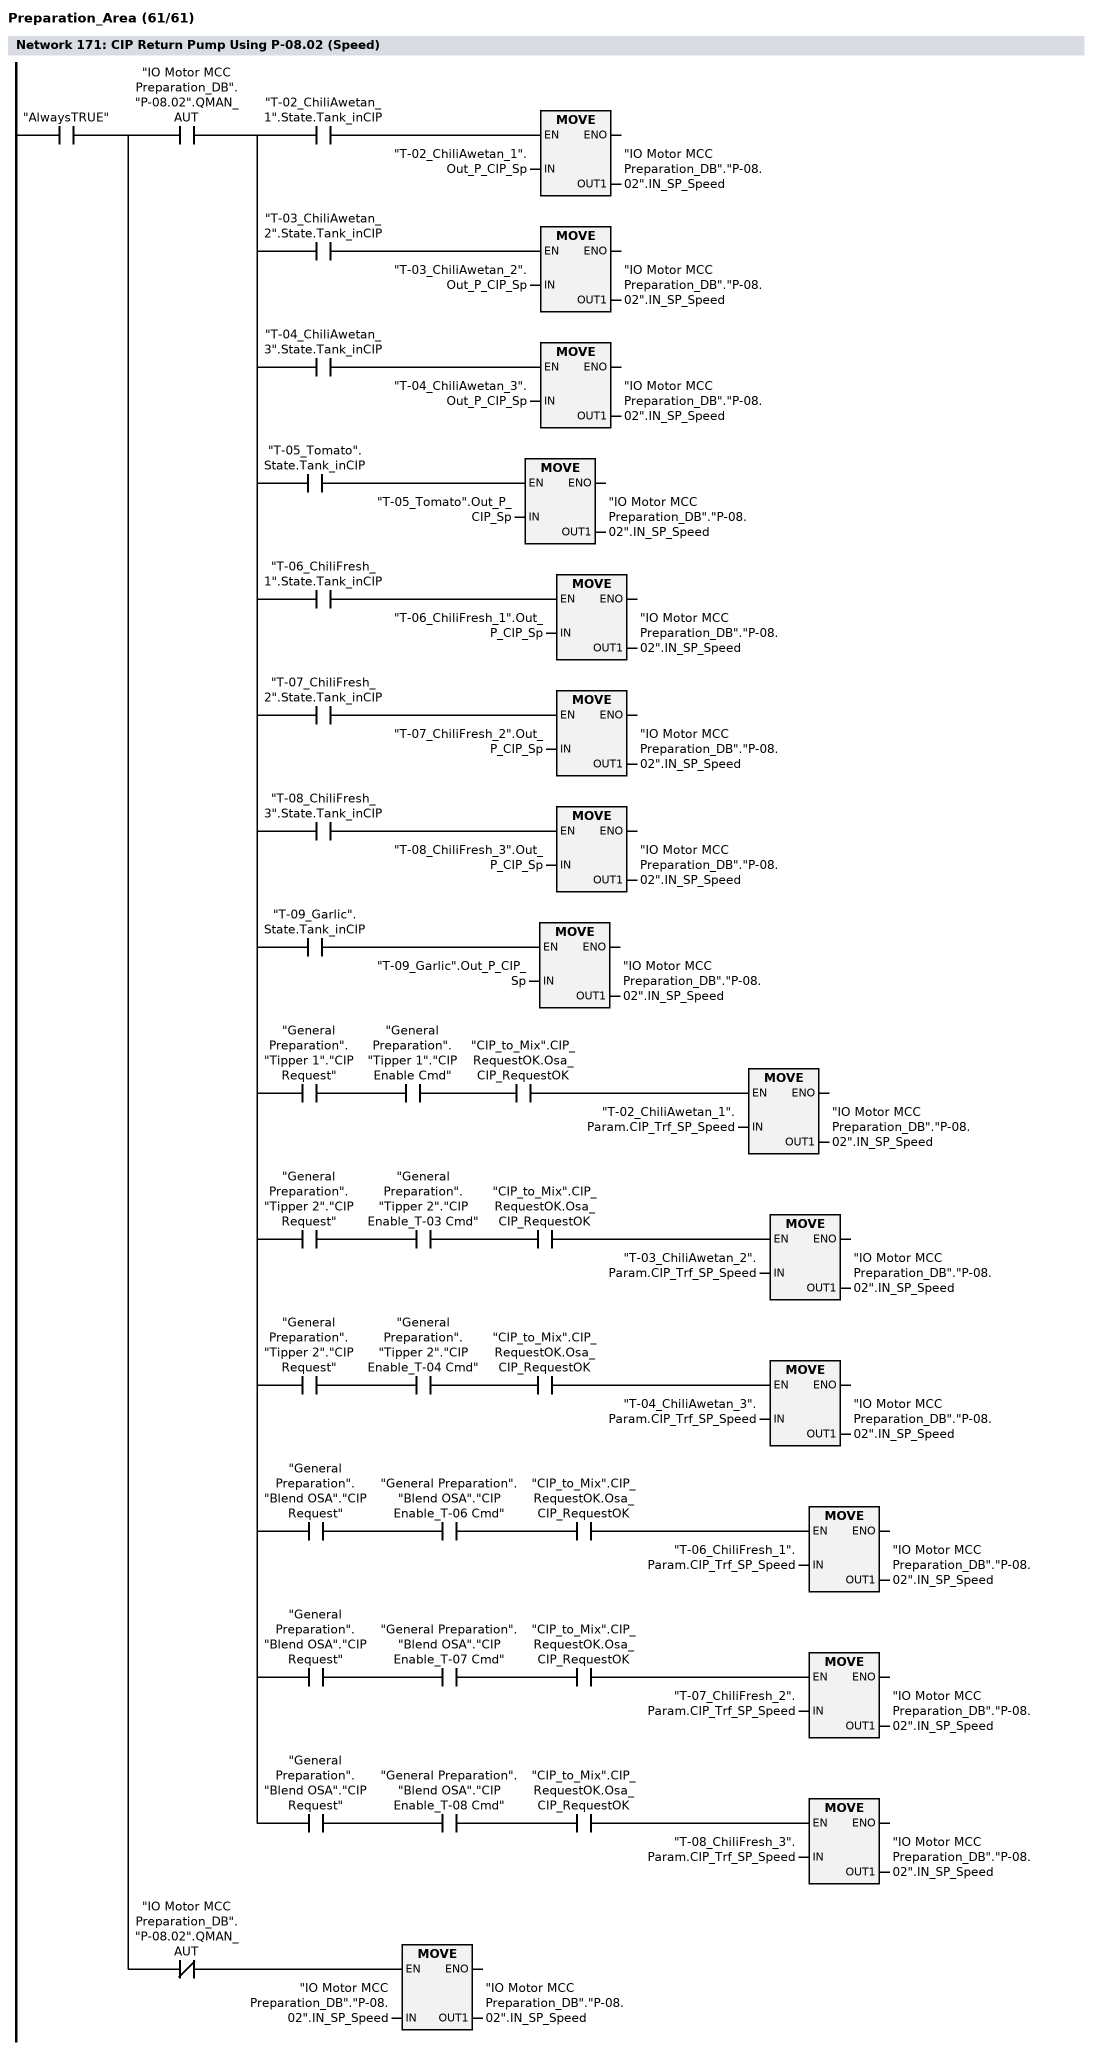
   RUNG wire#powerrail
      Contact( "AlwaysTRUE" )
      wire#w1
      Contact( "IO Motor MCC Preparation_DB"."P-08.02".QMAN_AUT )
      wire#w2
      Contact( "T-02_ChiliAwetan_1".State.Tank_inCIP )
      Move(in := "T-02_ChiliAwetan_1".Out_P_CIP_Sp, out1 => "IO Motor MCC Preparation_DB"."P-08.02".IN_SP_Speed)
   END_RUNG
   RUNG wire#w2
      Contact( "T-03_ChiliAwetan_2".State.Tank_inCIP )
      Move(in := "T-03_ChiliAwetan_2".Out_P_CIP_Sp, out1 => "IO Motor MCC Preparation_DB"."P-08.02".IN_SP_Speed)
   END_RUNG
   RUNG wire#w2
      Contact( "T-04_ChiliAwetan_3".State.Tank_inCIP )
      Move(in := "T-04_ChiliAwetan_3".Out_P_CIP_Sp, out1 => "IO Motor MCC Preparation_DB"."P-08.02".IN_SP_Speed)
   END_RUNG
   RUNG wire#w2
      Contact( "T-05_Tomato".State.Tank_inCIP )
      Move(in := "T-05_Tomato".Out_P_CIP_Sp, out1 => "IO Motor MCC Preparation_DB"."P-08.02".IN_SP_Speed)
   END_RUNG
   RUNG wire#w2
      Contact( "T-06_ChiliFresh_1".State.Tank_inCIP )
      Move(in := "T-06_ChiliFresh_1".Out_P_CIP_Sp, out1 => "IO Motor MCC Preparation_DB"."P-08.02".IN_SP_Speed)
   END_RUNG
   RUNG wire#w2
      Contact( "T-07_ChiliFresh_2".State.Tank_inCIP )
      Move(in := "T-07_ChiliFresh_2".Out_P_CIP_Sp, out1 => "IO Motor MCC Preparation_DB"."P-08.02".IN_SP_Speed)
   END_RUNG
   RUNG wire#w2
      Contact( "T-08_ChiliFresh_3".State.Tank_inCIP )
      Move(in := "T-08_ChiliFresh_3".Out_P_CIP_Sp, out1 => "IO Motor MCC Preparation_DB"."P-08.02".IN_SP_Speed)
   END_RUNG
   RUNG wire#w2
      Contact( "T-09_Garlic".State.Tank_inCIP )
      Move(in := "T-09_Garlic".Out_P_CIP_Sp, out1 => "IO Motor MCC Preparation_DB"."P-08.02".IN_SP_Speed)
   END_RUNG
   RUNG wire#w2
      Contact( "General Preparation"."Tipper 1"."CIP Request" )
      Contact( "General Preparation"."Tipper 1"."CIP Enable Cmd" )
      Contact( "CIP_to_Mix".CIP_RequestOK.Osa_CIP_RequestOK )
      Move(in := "T-02_ChiliAwetan_1".Param.CIP_Trf_SP_Speed, out1 => "IO Motor MCC Preparation_DB"."P-08.02".IN_SP_Speed)
   END_RUNG
   RUNG wire#w2
      Contact( "General Preparation"."Tipper 2"."CIP Request" )
      Contact( "General Preparation"."Tipper 2"."CIP Enable_T-03 Cmd" )
      Contact( "CIP_to_Mix".CIP_RequestOK.Osa_CIP_RequestOK )
      Move(in := "T-03_ChiliAwetan_2".Param.CIP_Trf_SP_Speed, out1 => "IO Motor MCC Preparation_DB"."P-08.02".IN_SP_Speed)
   END_RUNG
   RUNG wire#w2
      Contact( "General Preparation"."Tipper 2"."CIP Request" )
      Contact( "General Preparation"."Tipper 2"."CIP Enable_T-04 Cmd" )
      Contact( "CIP_to_Mix".CIP_RequestOK.Osa_CIP_RequestOK )
      Move(in := "T-04_ChiliAwetan_3".Param.CIP_Trf_SP_Speed, out1 => "IO Motor MCC Preparation_DB"."P-08.02".IN_SP_Speed)
   END_RUNG
   RUNG wire#w2
      Contact( "General Preparation"."Blend OSA"."CIP Request" )
      Contact( "General Preparation"."Blend OSA"."CIP Enable_T-06 Cmd" )
      Contact( "CIP_to_Mix".CIP_RequestOK.Osa_CIP_RequestOK )
      Move(in := "T-06_ChiliFresh_1".Param.CIP_Trf_SP_Speed, out1 => "IO Motor MCC Preparation_DB"."P-08.02".IN_SP_Speed)
   END_RUNG
   RUNG wire#w2
      Contact( "General Preparation"."Blend OSA"."CIP Request" )
      Contact( "General Preparation"."Blend OSA"."CIP Enable_T-07 Cmd" )
      Contact( "CIP_to_Mix".CIP_RequestOK.Osa_CIP_RequestOK )
      Move(in := "T-07_ChiliFresh_2".Param.CIP_Trf_SP_Speed, out1 => "IO Motor MCC Preparation_DB"."P-08.02".IN_SP_Speed)
   END_RUNG
   RUNG wire#w2
      Contact( "General Preparation"."Blend OSA"."CIP Request" )
      Contact( "General Preparation"."Blend OSA"."CIP Enable_T-08 Cmd" )
      Contact( "CIP_to_Mix".CIP_RequestOK.Osa_CIP_RequestOK )
      Move(in := "T-08_ChiliFresh_3".Param.CIP_Trf_SP_Speed, out1 => "IO Motor MCC Preparation_DB"."P-08.02".IN_SP_Speed)
   END_RUNG
   RUNG wire#w1
      I_Contact( "IO Motor MCC Preparation_DB"."P-08.02".QMAN_AUT )
      Move(in := "IO Motor MCC Preparation_DB"."P-08.02".IN_SP_Speed, out1 => "IO Motor MCC Preparation_DB"."P-08.02".IN_SP_Speed)
   END_RUNG
   // the same network as SCL:
   #_w1 := "AlwaysTRUE" AND "IO Motor MCC Preparation_DB"."P-08.02".QMAN_AUT;
   IF #_w1 AND "T-02_ChiliAwetan_1".State.Tank_inCIP THEN
       "IO Motor MCC Preparation_DB"."P-08.02".IN_SP_Speed := "T-02_ChiliAwetan_1".Out_P_CIP_Sp;
   END_IF;
   IF #_w1 AND "T-03_ChiliAwetan_2".State.Tank_inCIP THEN
       "IO Motor MCC Preparation_DB"."P-08.02".IN_SP_Speed := "T-03_ChiliAwetan_2".Out_P_CIP_Sp;
   END_IF;
   IF #_w1 AND "T-04_ChiliAwetan_3".State.Tank_inCIP THEN
       "IO Motor MCC Preparation_DB"."P-08.02".IN_SP_Speed := "T-04_ChiliAwetan_3".Out_P_CIP_Sp;
   END_IF;
   IF #_w1 AND "T-05_Tomato".State.Tank_inCIP THEN
       "IO Motor MCC Preparation_DB"."P-08.02".IN_SP_Speed := "T-05_Tomato".Out_P_CIP_Sp;
   END_IF;
   IF #_w1 AND "T-06_ChiliFresh_1".State.Tank_inCIP THEN
       "IO Motor MCC Preparation_DB"."P-08.02".IN_SP_Speed := "T-06_ChiliFresh_1".Out_P_CIP_Sp;
   END_IF;
   IF #_w1 AND "T-07_ChiliFresh_2".State.Tank_inCIP THEN
       "IO Motor MCC Preparation_DB"."P-08.02".IN_SP_Speed := "T-07_ChiliFresh_2".Out_P_CIP_Sp;
   END_IF;
   IF #_w1 AND "T-08_ChiliFresh_3".State.Tank_inCIP THEN
       "IO Motor MCC Preparation_DB"."P-08.02".IN_SP_Speed := "T-08_ChiliFresh_3".Out_P_CIP_Sp;
   END_IF;
   IF #_w1 AND "T-09_Garlic".State.Tank_inCIP THEN
       "IO Motor MCC Preparation_DB"."P-08.02".IN_SP_Speed := "T-09_Garlic".Out_P_CIP_Sp;
   END_IF;
   IF #_w1 AND "General Preparation"."Tipper 1"."CIP Request" AND "General Preparation"."Tipper 1"."CIP Enable Cmd" AND "CIP_to_Mix".CIP_RequestOK.Osa_CIP_RequestOK THEN
       "IO Motor MCC Preparation_DB"."P-08.02".IN_SP_Speed := "T-02_ChiliAwetan_1".Param.CIP_Trf_SP_Speed;
   END_IF;
   IF #_w1 AND "General Preparation"."Tipper 2"."CIP Request" AND "General Preparation"."Tipper 2"."CIP Enable_T-03 Cmd" AND "CIP_to_Mix".CIP_RequestOK.Osa_CIP_RequestOK THEN
       "IO Motor MCC Preparation_DB"."P-08.02".IN_SP_Speed := "T-03_ChiliAwetan_2".Param.CIP_Trf_SP_Speed;
   END_IF;
   IF #_w1 AND "General Preparation"."Tipper 2"."CIP Request" AND "General Preparation"."Tipper 2"."CIP Enable_T-04 Cmd" AND "CIP_to_Mix".CIP_RequestOK.Osa_CIP_RequestOK THEN
       "IO Motor MCC Preparation_DB"."P-08.02".IN_SP_Speed := "T-04_ChiliAwetan_3".Param.CIP_Trf_SP_Speed;
   END_IF;
   IF #_w1 AND "General Preparation"."Blend OSA"."CIP Request" AND "General Preparation"."Blend OSA"."CIP Enable_T-06 Cmd" AND "CIP_to_Mix".CIP_RequestOK.Osa_CIP_RequestOK THEN
       "IO Motor MCC Preparation_DB"."P-08.02".IN_SP_Speed := "T-06_ChiliFresh_1".Param.CIP_Trf_SP_Speed;
   END_IF;
   IF #_w1 AND "General Preparation"."Blend OSA"."CIP Request" AND "General Preparation"."Blend OSA"."CIP Enable_T-07 Cmd" AND "CIP_to_Mix".CIP_RequestOK.Osa_CIP_RequestOK THEN
       "IO Motor MCC Preparation_DB"."P-08.02".IN_SP_Speed := "T-07_ChiliFresh_2".Param.CIP_Trf_SP_Speed;
   END_IF;
   IF #_w1 AND "General Preparation"."Blend OSA"."CIP Request" AND "General Preparation"."Blend OSA"."CIP Enable_T-08 Cmd" AND "CIP_to_Mix".CIP_RequestOK.Osa_CIP_RequestOK THEN
       "IO Motor MCC Preparation_DB"."P-08.02".IN_SP_Speed := "T-08_ChiliFresh_3".Param.CIP_Trf_SP_Speed;
   END_IF;
   IF "AlwaysTRUE" AND NOT "IO Motor MCC Preparation_DB"."P-08.02".QMAN_AUT THEN
       "IO Motor MCC Preparation_DB"."P-08.02".IN_SP_Speed := "IO Motor MCC Preparation_DB"."P-08.02".IN_SP_Speed;
   END_IF;
END_REGION

NETWORK
TITLE = Valve IO
//Valve T-02.01 Chili Awetan Tank 1
      CALL  "IO Valve T02 Chili", "IO_Valve_T02_Chili"
      ( lock    := ,
        Init    := "General_DB".Initial,
        testing := "General_DB"."Testing FB Valve".Preparation,
        Reset   := "General_DB".Reset
      );
//Valve T-03.01 Chili Awetan Tank 2
      CALL  "IO Valve T03 Chili", "IO_Valve_T03_Chili"
      ( lock    := ,
        Init    := "General_DB".Initial,
        testing := "General_DB"."Testing FB Valve".Preparation,
        Reset   := "General_DB".Reset
      );
//Valve T-04.01 Chili Awetan Tank 3
      CALL  "IO Valve T04 Chili", "IO_Valve_T04_Chili"
      ( lock    := ,
        Init    := "General_DB".Initial,
        testing := "General_DB"."Testing FB Valve".Preparation,
        Reset   := "General_DB".Reset
      );
//Valve T-05.01 Tomato Tank
      CALL  "IO Valve T05 Tomato", "IO_Valve_T05_Tomato"
      ( lock    := ,
        Init    := "General_DB".Initial,
        testing := "General_DB"."Testing FB Valve".Preparation,
        Reset   := "General_DB".Reset
      );
//Valve T-06.01 Fresh Chili Tank 1
      CALL  "IO Valve T06 FreshChili", "IO_Valve_T06_FreshChili"
      ( lock    := ,
        Init    := "General_DB".Initial,
        testing := "General_DB"."Testing FB Valve".Preparation,
        Reset   := "General_DB".Reset
      );
//Valve T-07.01 Fresh Chili Tank 2
      CALL  "IO Valve T07 FreshChili", "IO_Valve_T07_FreshChili"
      ( lock    := ,
        Init    := "General_DB".Initial,
        testing := "General_DB"."Testing FB Valve".Preparation,
        Reset   := "General_DB".Reset
      );
//Valve T-08.01 Fresh Chili Tank 3
      CALL  "IO Valve T08 FreshChili", "IO_Valve_T08_FreshChili"
      ( lock    := ,
        Init    := "General_DB".Initial,
        testing := "General_DB"."Testing FB Valve".Preparation,
        Reset   := "General_DB".Reset
      );
//Valve T-09.01 Garlic Tank
      CALL  "IO Valve T09 Garlic", "IO_Valve_T09_Garlic"
      ( lock    := ,
        Init    := "General_DB".Initial,
        testing := "General_DB"."Testing FB Valve".Preparation,
        Reset   := "General_DB".Reset
      );
//Valve T-10.01 Vinegar Tank
      CALL  "IO Valve T10 Vinegar", "IO_Valve_T10_Vinegar"
      ( lock    := ,
        Init    := "General_DB".Initial,
        testing := "General_DB"."Testing FB Valve".Preparation,
        Reset   := "General_DB".Reset
      );
//Valve T-10.01 HotWater
      CALL  "IO Valve T51 HotWaterLine", "IO_Valve_T51_HW"
      ( lock    := ,
        Init    := "General_DB".Initial,
        testing := "General_DB"."Testing FB Valve".Preparation,
        Reset   := "General_DB".Reset
      );


END_FUNCTION
